// TIA Portal V20 export
FUNCTION_BLOCK "Sequence_3_JellyRollWinder"   // FB224, LAD
AUTHOR : ERsystem_FA2_DH. Kim
// stored: IsIECCheckEnabled true, MemoryReserve 100, Namespace Unit1.Em7, SetENOAutomatically false
   VAR
      statSelectedJobNumber { ExternalWritable := 'False'} : DInt;   // Evaluated Job Number
      instSequenceLADStatus { ExternalWritable := 'False'} : "LAF_StatusLadSequence";
      instSequenceLADControl { ExternalWritable := 'False'} : "LAF_ControlLadSequence";
      statTonTime { ExternalAccessible := 'False'; ExternalVisible := 'False'; ExternalWritable := 'False'} : Array[0..999] of TON_TIME;
   END_VAR
   VAR_TEMP
      tempCustomerAction : Bool;   // Placeholder for possible actions
      tempDo_nothing_and_wait_for_init : Bool;   // Placeholder for doing nothing
      tempSafeStateCondition : Bool;   // Temp Condition for the equipment module to be in a safe state
      tempIndex : Int;
   END_VAR
   VAR CONSTANT
      STEP_IDLE : DInt := 1;
      STEP_IMMEDIATE_STOP : DInt := 9001;   // Step executed when an immediate stop command is triggered for the sequence (i.e. when unit is in state aborting)
      JOB_1_STEP_01 : DInt := 101;
      JOB_1_STEP_10 : DInt := 110;
      JOB_1_STEP_20 : DInt := 120;
      JOB_1_STEP_30 : DInt := 130;
      JOB_1_STEP_80 : DInt := 180;
      JOB_1_STEP_90 : DInt := 190;
      JOB_2_STEP_01 : DInt := 201;
      JOB_2_STEP_10 : DInt := 210;
      JOB_2_STEP_20 : DInt := 220;
      JOB_2_STEP_21 : DInt := 221;
      JOB_2_STEP_90 : DInt := 290;
      JOB_3_STEP_01 : DInt := 301;
      JOB_3_STEP_10 : DInt := 310;
      JOB_3_STEP_11 : DInt := 311;
      JOB_3_STEP_12 : DInt := 312;
      JOB_3_STEP_13 : DInt := 313;
      JOB_3_STEP_90 : DInt := 390;
      JOB_4_STEP_01 : DInt := 401;
      JOB_4_STEP_10 : DInt := 410;
      JOB_4_STEP_20 : DInt := 420;
      JOB_4_STEP_21 : DInt := 421;
      JOB_4_STEP_90 : DInt := 490;
      JOB_5_STEP_01 : DInt := 501;
      JOB_5_STEP_10 : DInt := 510;
      JOB_5_STEP_11 : DInt := 511;
      JOB_5_STEP_20 : DInt := 520;
      JOB_5_STEP_21 : DInt := 521;
      JOB_5_STEP_90 : DInt := 590;
      JOB_6_STEP_01 : DInt := 601;
      JOB_6_STEP_10 : DInt := 610;
      JOB_6_STEP_20 : DInt := 620;
      JOB_6_STEP_21 : DInt := 621;
      JOB_6_STEP_30 : DInt := 630;
      JOB_6_STEP_80 : DInt := 680;
      JOB_6_STEP_81 : DInt := 681;
      JOB_6_STEP_90 : DInt := 690;
      JOB_7_STEP_01 : DInt := 701;
      JOB_7_STEP_10 : DInt := 710;
      JOB_7_STEP_20 : DInt := 720;
      JOB_7_STEP_30 : DInt := 730;
      JOB_7_STEP_40 : DInt := 740;
      JOB_7_STEP_50 : DInt := 750;
      JOB_7_STEP_90 : DInt := 790;
      JOB_10_STEP_01 : DInt := 1001;
      JOB_10_STEP_10 : DInt := 1010;
      JOB_10_STEP_90 : DInt := 1090;
      JOB_11_STEP_01 : DInt := 1101;
      JOB_11_STEP_10 : DInt := 1110;
      JOB_11_STEP_20 : DInt := 1120;
      JOB_11_STEP_90 : DInt := 1190;
      JOB_12_STEP_01 : DInt := 1201;
      JOB_12_STEP_10 : DInt := 1210;
      JOB_12_STEP_11 : DInt := 1211;
      JOB_12_STEP_90 : DInt := 1290;
      JOB_13_STEP_01 : DInt := 1301;
      JOB_13_STEP_10 : DInt := 1310;
      JOB_13_STEP_90 : DInt := 1390;
      JOB_14_STEP_01 : DInt := 1401;
      JOB_14_STEP_10 : DInt := 1410;
      JOB_14_STEP_90 : DInt := 1490;
      FALSE : Bool := FALSE;
      TRUE : Bool := TRUE;
   END_VAR
   VAR_TEMP   // added for the SCL form of the ladder/FBD networks
      _w1 : Bool;
      _w2 : Bool;
   END_VAR
BEGIN

REGION Network 1: BLOCK INFO HEADER
   // (company) / (C) Copyright (year)
   // ---------------------------------------------------------------------------------
   // Title:                             (Title of this block)
   // Comment/Function: (that is implemented in the block)
   // Library/Family:           (that the source is dedicated to)
   // Author:                        (department / person in charge / contact)
   // Target System:          (test system with FW version)
   // Engineering:              TIA Portal (SW version)
   // Restrictions:               (OB types, etc.)
   // Requirements:           (hardware, technological package, etc.)
   // ---------------------------------------------------------------------------------
   // Change log table:
   // Version          | Date             | Signature      | Expert in charge  | Changes applied ------------------------|----------------------|-------------------------|--------------------------------|-----------------------
   // 001.000.000 | yyyy-mm-dd | 0x00000000 | (name of expert) | First released version
END_REGION

REGION Network 2: DESCRIPTION
   // This is a template block provided by the Automation Framework. It can be used to create an own project.
   // The Block Info Header is prepared to put in your own data.
   // Description of the block could be added here and the docu created by Code2Docu.
END_REGION

REGION Network 3: ********************* CONTROL *************************
END_REGION

REGION Network 4: Sequence Control
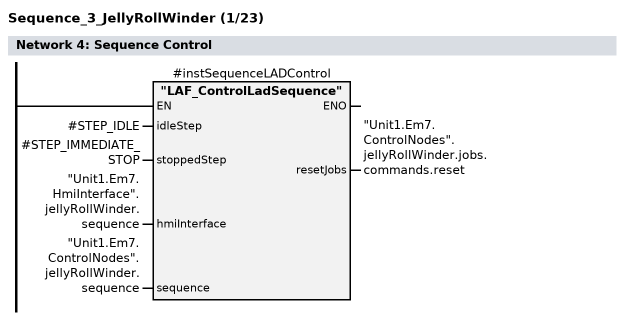
   RUNG wire#powerrail
      #instSequenceLADControl(idleStep := #STEP_IDLE, stoppedStep := #STEP_IMMEDIATE_STOP, hmiInterface := "Unit1.Em7.HmiInterface".jellyRollWinder.sequence, sequence := "Unit1.Em7.ControlNodes".jellyRollWinder.sequence, resetJobs => "Unit1.Em7.ControlNodes".jellyRollWinder.jobs.commands.reset)
   END_RUNG
   // the same network as SCL:
   #instSequenceLADControl(idleStep := #STEP_IDLE,   // "LAF_ControlLadSequence"
                           stoppedStep := #STEP_IMMEDIATE_STOP,
                           hmiInterface := "Unit1.Em7.HmiInterface".jellyRollWinder.sequence,
                           sequence := "Unit1.Em7.ControlNodes".jellyRollWinder.sequence,
                           resetJobs => "Unit1.Em7.ControlNodes".jellyRollWinder.jobs.commands.reset);
END_REGION

REGION Network 5: *************** JOB SELECT **************************
END_REGION

REGION Network 6: STEP IDLE
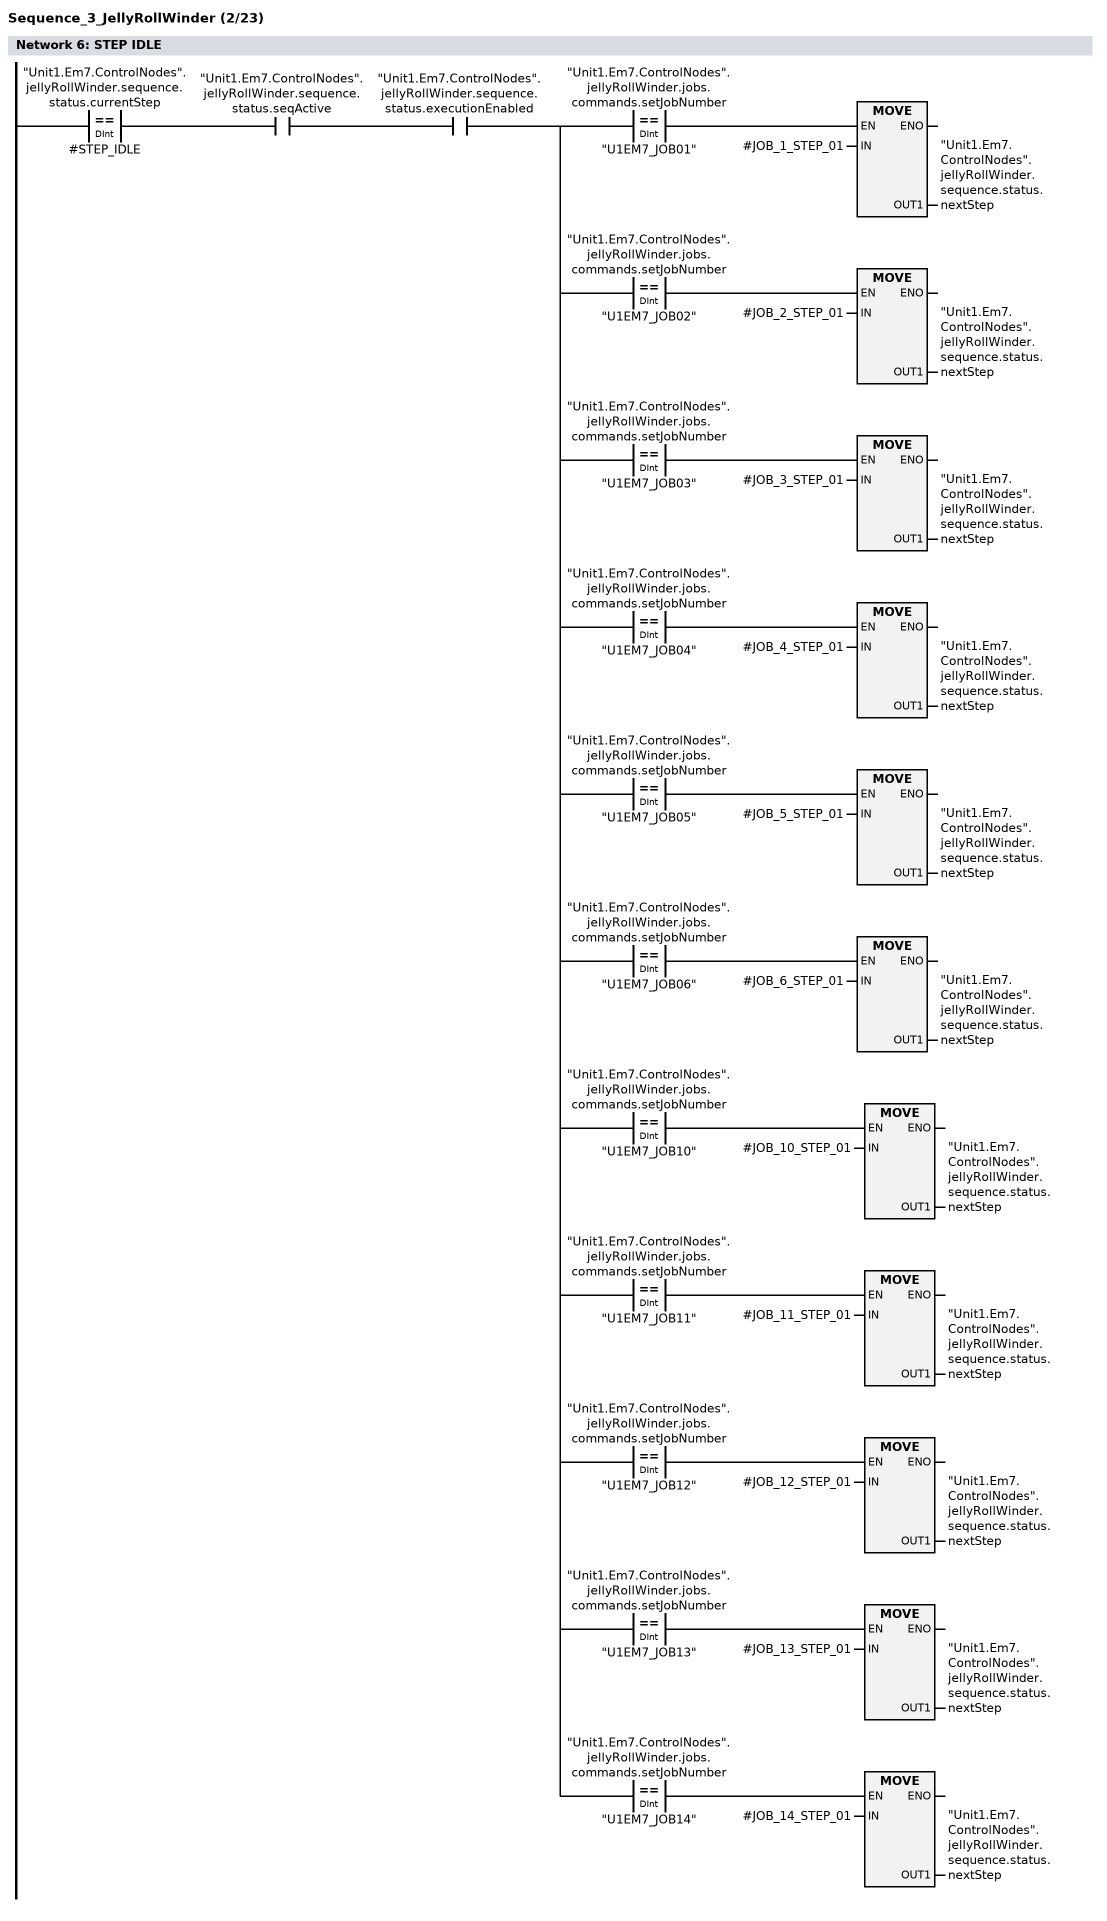
   RUNG wire#powerrail
      { S7_Templates := "SrcType := DInt" } EQ_Contact(in1 := "Unit1.Em7.ControlNodes".jellyRollWinder.sequence.status.currentStep, in2 := #STEP_IDLE)
      Contact( "Unit1.Em7.ControlNodes".jellyRollWinder.sequence.status.seqActive )
      Contact( "Unit1.Em7.ControlNodes".jellyRollWinder.sequence.status.executionEnabled )
      wire#w1
      { S7_Templates := "SrcType := DInt" } EQ_Contact(in1 := "Unit1.Em7.ControlNodes".jellyRollWinder.jobs.commands.setJobNumber, in2 := "U1EM7_JOB01")
      Move(in := #JOB_1_STEP_01, out1 => "Unit1.Em7.ControlNodes".jellyRollWinder.sequence.status.nextStep)
   END_RUNG
   RUNG wire#w1
      { S7_Templates := "SrcType := DInt" } EQ_Contact(in1 := "Unit1.Em7.ControlNodes".jellyRollWinder.jobs.commands.setJobNumber, in2 := "U1EM7_JOB02")
      Move(in := #JOB_2_STEP_01, out1 => "Unit1.Em7.ControlNodes".jellyRollWinder.sequence.status.nextStep)
   END_RUNG
   RUNG wire#w1
      { S7_Templates := "SrcType := DInt" } EQ_Contact(in1 := "Unit1.Em7.ControlNodes".jellyRollWinder.jobs.commands.setJobNumber, in2 := "U1EM7_JOB03")
      Move(in := #JOB_3_STEP_01, out1 => "Unit1.Em7.ControlNodes".jellyRollWinder.sequence.status.nextStep)
   END_RUNG
   RUNG wire#w1
      { S7_Templates := "SrcType := DInt" } EQ_Contact(in1 := "Unit1.Em7.ControlNodes".jellyRollWinder.jobs.commands.setJobNumber, in2 := "U1EM7_JOB04")
      Move(in := #JOB_4_STEP_01, out1 => "Unit1.Em7.ControlNodes".jellyRollWinder.sequence.status.nextStep)
   END_RUNG
   RUNG wire#w1
      { S7_Templates := "SrcType := DInt" } EQ_Contact(in1 := "Unit1.Em7.ControlNodes".jellyRollWinder.jobs.commands.setJobNumber, in2 := "U1EM7_JOB05")
      Move(in := #JOB_5_STEP_01, out1 => "Unit1.Em7.ControlNodes".jellyRollWinder.sequence.status.nextStep)
   END_RUNG
   RUNG wire#w1
      { S7_Templates := "SrcType := DInt" } EQ_Contact(in1 := "Unit1.Em7.ControlNodes".jellyRollWinder.jobs.commands.setJobNumber, in2 := "U1EM7_JOB06")
      Move(in := #JOB_6_STEP_01, out1 => "Unit1.Em7.ControlNodes".jellyRollWinder.sequence.status.nextStep)
   END_RUNG
   RUNG wire#w1
      { S7_Templates := "SrcType := DInt" } EQ_Contact(in1 := "Unit1.Em7.ControlNodes".jellyRollWinder.jobs.commands.setJobNumber, in2 := "U1EM7_JOB10")
      Move(in := #JOB_10_STEP_01, out1 => "Unit1.Em7.ControlNodes".jellyRollWinder.sequence.status.nextStep)
   END_RUNG
   RUNG wire#w1
      { S7_Templates := "SrcType := DInt" } EQ_Contact(in1 := "Unit1.Em7.ControlNodes".jellyRollWinder.jobs.commands.setJobNumber, in2 := "U1EM7_JOB11")
      Move(in := #JOB_11_STEP_01, out1 => "Unit1.Em7.ControlNodes".jellyRollWinder.sequence.status.nextStep)
   END_RUNG
   RUNG wire#w1
      { S7_Templates := "SrcType := DInt" } EQ_Contact(in1 := "Unit1.Em7.ControlNodes".jellyRollWinder.jobs.commands.setJobNumber, in2 := "U1EM7_JOB12")
      Move(in := #JOB_12_STEP_01, out1 => "Unit1.Em7.ControlNodes".jellyRollWinder.sequence.status.nextStep)
   END_RUNG
   RUNG wire#w1
      { S7_Templates := "SrcType := DInt" } EQ_Contact(in1 := "Unit1.Em7.ControlNodes".jellyRollWinder.jobs.commands.setJobNumber, in2 := "U1EM7_JOB13")
      Move(in := #JOB_13_STEP_01, out1 => "Unit1.Em7.ControlNodes".jellyRollWinder.sequence.status.nextStep)
   END_RUNG
   RUNG wire#w1
      { S7_Templates := "SrcType := DInt" } EQ_Contact(in1 := "Unit1.Em7.ControlNodes".jellyRollWinder.jobs.commands.setJobNumber, in2 := "U1EM7_JOB14")
      Move(in := #JOB_14_STEP_01, out1 => "Unit1.Em7.ControlNodes".jellyRollWinder.sequence.status.nextStep)
   END_RUNG
   // the same network as SCL:
   #_w1 := ("Unit1.Em7.ControlNodes".jellyRollWinder.sequence.status.currentStep = #STEP_IDLE) AND "Unit1.Em7.ControlNodes".jellyRollWinder.sequence.status.seqActive AND "Unit1.Em7.ControlNodes".jellyRollWinder.sequence.status.executionEnabled;
   IF #_w1 AND ("Unit1.Em7.ControlNodes".jellyRollWinder.jobs.commands.setJobNumber = "U1EM7_JOB01") THEN
       "Unit1.Em7.ControlNodes".jellyRollWinder.sequence.status.nextStep := #JOB_1_STEP_01;
   END_IF;
   IF #_w1 AND ("Unit1.Em7.ControlNodes".jellyRollWinder.jobs.commands.setJobNumber = "U1EM7_JOB02") THEN
       "Unit1.Em7.ControlNodes".jellyRollWinder.sequence.status.nextStep := #JOB_2_STEP_01;
   END_IF;
   IF #_w1 AND ("Unit1.Em7.ControlNodes".jellyRollWinder.jobs.commands.setJobNumber = "U1EM7_JOB03") THEN
       "Unit1.Em7.ControlNodes".jellyRollWinder.sequence.status.nextStep := #JOB_3_STEP_01;
   END_IF;
   IF #_w1 AND ("Unit1.Em7.ControlNodes".jellyRollWinder.jobs.commands.setJobNumber = "U1EM7_JOB04") THEN
       "Unit1.Em7.ControlNodes".jellyRollWinder.sequence.status.nextStep := #JOB_4_STEP_01;
   END_IF;
   IF #_w1 AND ("Unit1.Em7.ControlNodes".jellyRollWinder.jobs.commands.setJobNumber = "U1EM7_JOB05") THEN
       "Unit1.Em7.ControlNodes".jellyRollWinder.sequence.status.nextStep := #JOB_5_STEP_01;
   END_IF;
   IF #_w1 AND ("Unit1.Em7.ControlNodes".jellyRollWinder.jobs.commands.setJobNumber = "U1EM7_JOB06") THEN
       "Unit1.Em7.ControlNodes".jellyRollWinder.sequence.status.nextStep := #JOB_6_STEP_01;
   END_IF;
   IF #_w1 AND ("Unit1.Em7.ControlNodes".jellyRollWinder.jobs.commands.setJobNumber = "U1EM7_JOB10") THEN
       "Unit1.Em7.ControlNodes".jellyRollWinder.sequence.status.nextStep := #JOB_10_STEP_01;
   END_IF;
   IF #_w1 AND ("Unit1.Em7.ControlNodes".jellyRollWinder.jobs.commands.setJobNumber = "U1EM7_JOB11") THEN
       "Unit1.Em7.ControlNodes".jellyRollWinder.sequence.status.nextStep := #JOB_11_STEP_01;
   END_IF;
   IF #_w1 AND ("Unit1.Em7.ControlNodes".jellyRollWinder.jobs.commands.setJobNumber = "U1EM7_JOB12") THEN
       "Unit1.Em7.ControlNodes".jellyRollWinder.sequence.status.nextStep := #JOB_12_STEP_01;
   END_IF;
   IF #_w1 AND ("Unit1.Em7.ControlNodes".jellyRollWinder.jobs.commands.setJobNumber = "U1EM7_JOB13") THEN
       "Unit1.Em7.ControlNodes".jellyRollWinder.sequence.status.nextStep := #JOB_13_STEP_01;
   END_IF;
   IF #_w1 AND ("Unit1.Em7.ControlNodes".jellyRollWinder.jobs.commands.setJobNumber = "U1EM7_JOB14") THEN
       "Unit1.Em7.ControlNodes".jellyRollWinder.sequence.status.nextStep := #JOB_14_STEP_01;
   END_IF;
END_REGION

REGION Network 7: ******************** JOB[1] EM HOMING ********************
END_REGION

REGION Network 8: Step[101] : JOB[1] Condition
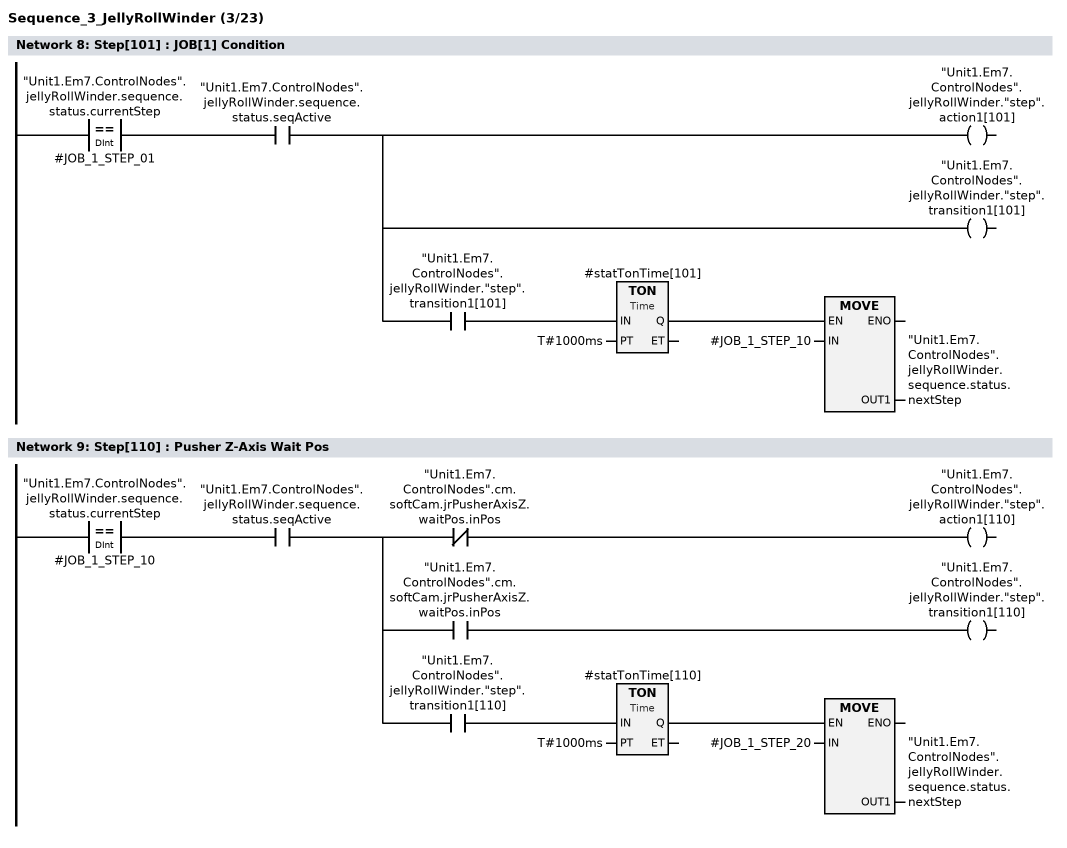
   RUNG wire#powerrail
      { S7_Templates := "SrcType := DInt" } EQ_Contact(in1 := "Unit1.Em7.ControlNodes".jellyRollWinder.sequence.status.currentStep, in2 := #JOB_1_STEP_01)
      Contact( "Unit1.Em7.ControlNodes".jellyRollWinder.sequence.status.seqActive )
      wire#w1
      Coil( "Unit1.Em7.ControlNodes".jellyRollWinder."step".action1[101] )
   END_RUNG
   RUNG wire#w1
      Coil( "Unit1.Em7.ControlNodes".jellyRollWinder."step".transition1[101] )
   END_RUNG
   RUNG wire#w1
      Contact( "Unit1.Em7.ControlNodes".jellyRollWinder."step".transition1[101] )
      { S7_Templates := "time_type := Time" } #statTonTime[101].TON(pt := T#1000ms, et =>)
      Move(in := #JOB_1_STEP_10, out1 => "Unit1.Em7.ControlNodes".jellyRollWinder.sequence.status.nextStep)
   END_RUNG
   // the same network as SCL:
   "Unit1.Em7.ControlNodes".jellyRollWinder."step".action1[101] := ("Unit1.Em7.ControlNodes".jellyRollWinder.sequence.status.currentStep = #JOB_1_STEP_01) AND "Unit1.Em7.ControlNodes".jellyRollWinder.sequence.status.seqActive;
   "Unit1.Em7.ControlNodes".jellyRollWinder."step".transition1[101] := ("Unit1.Em7.ControlNodes".jellyRollWinder.sequence.status.currentStep = #JOB_1_STEP_01) AND "Unit1.Em7.ControlNodes".jellyRollWinder.sequence.status.seqActive;
   #statTonTime[101].TON(IN := ("Unit1.Em7.ControlNodes".jellyRollWinder.sequence.status.currentStep = #JOB_1_STEP_01) AND "Unit1.Em7.ControlNodes".jellyRollWinder.sequence.status.seqActive AND "Unit1.Em7.ControlNodes".jellyRollWinder."step".transition1[101],
                         PT := T#1000ms);
   IF #statTonTime[101].Q THEN
       "Unit1.Em7.ControlNodes".jellyRollWinder.sequence.status.nextStep := #JOB_1_STEP_10;
   END_IF;
END_REGION

REGION Network 9: Step[110] : Pusher Z-Axis Wait Pos
   RUNG wire#powerrail
      { S7_Templates := "SrcType := DInt" } EQ_Contact(in1 := "Unit1.Em7.ControlNodes".jellyRollWinder.sequence.status.currentStep, in2 := #JOB_1_STEP_10)
      Contact( "Unit1.Em7.ControlNodes".jellyRollWinder.sequence.status.seqActive )
      wire#w1
      I_Contact( "Unit1.Em7.ControlNodes".cm.softCam.jrPusherAxisZ.waitPos.inPos )
      Coil( "Unit1.Em7.ControlNodes".jellyRollWinder."step".action1[110] )
   END_RUNG
   RUNG wire#w1
      Contact( "Unit1.Em7.ControlNodes".cm.softCam.jrPusherAxisZ.waitPos.inPos )
      Coil( "Unit1.Em7.ControlNodes".jellyRollWinder."step".transition1[110] )
   END_RUNG
   RUNG wire#w1
      Contact( "Unit1.Em7.ControlNodes".jellyRollWinder."step".transition1[110] )
      { S7_Templates := "time_type := Time" } #statTonTime[110].TON(pt := T#1000ms, et =>)
      Move(in := #JOB_1_STEP_20, out1 => "Unit1.Em7.ControlNodes".jellyRollWinder.sequence.status.nextStep)
   END_RUNG
   // the same network as SCL:
   #_w1 := ("Unit1.Em7.ControlNodes".jellyRollWinder.sequence.status.currentStep = #JOB_1_STEP_10) AND "Unit1.Em7.ControlNodes".jellyRollWinder.sequence.status.seqActive;
   "Unit1.Em7.ControlNodes".jellyRollWinder."step".action1[110] := #_w1 AND NOT "Unit1.Em7.ControlNodes".cm.softCam.jrPusherAxisZ.waitPos.inPos;
   "Unit1.Em7.ControlNodes".jellyRollWinder."step".transition1[110] := #_w1 AND "Unit1.Em7.ControlNodes".cm.softCam.jrPusherAxisZ.waitPos.inPos;
   #statTonTime[110].TON(IN := #_w1 AND "Unit1.Em7.ControlNodes".jellyRollWinder."step".transition1[110],
                         PT := T#1000ms);
   IF #statTonTime[110].Q THEN
       "Unit1.Em7.ControlNodes".jellyRollWinder.sequence.status.nextStep := #JOB_1_STEP_20;
   END_IF;
END_REGION

REGION Network 10: Step[120]: Pusher Backward
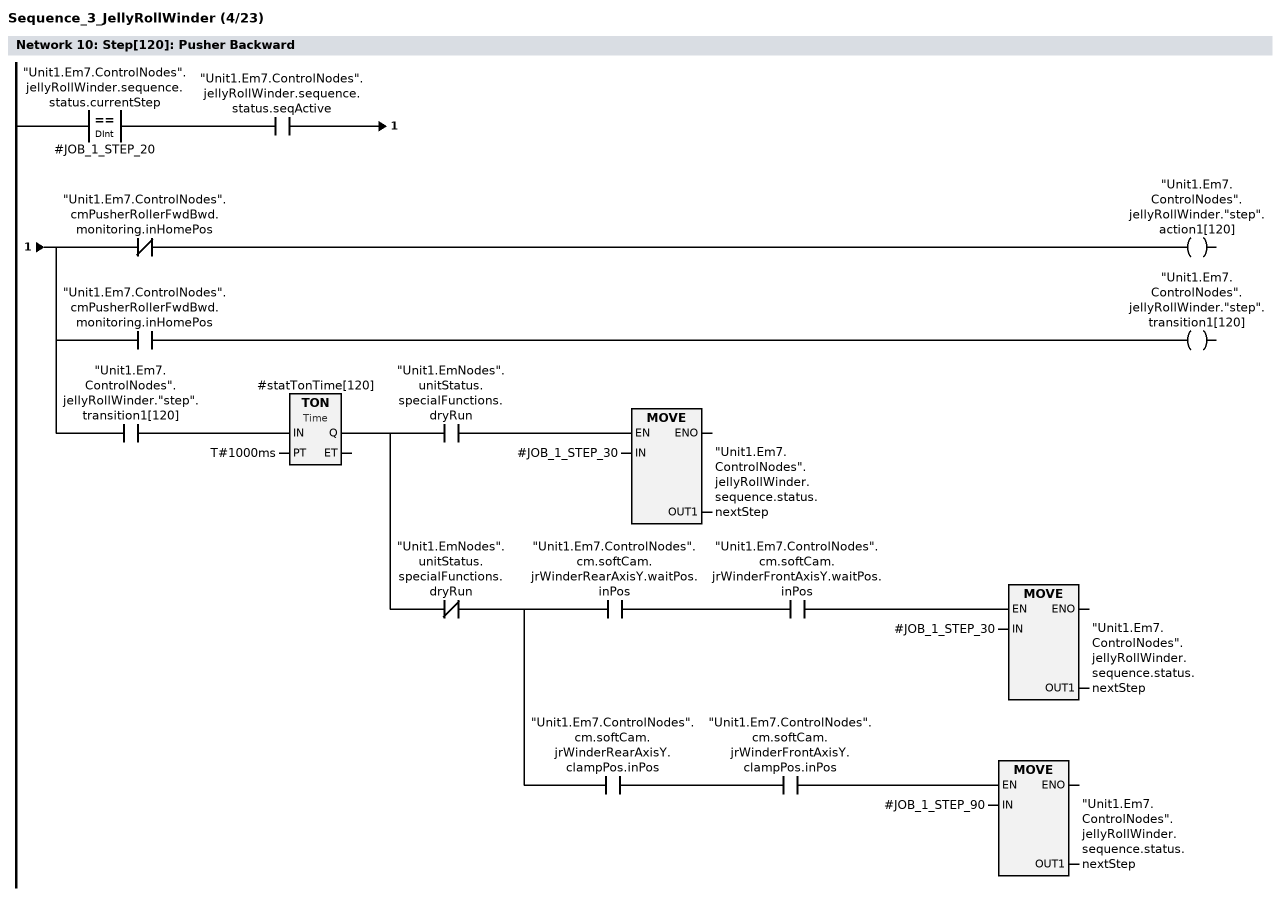
   RUNG wire#powerrail
      { S7_Templates := "SrcType := DInt" } EQ_Contact(in1 := "Unit1.Em7.ControlNodes".jellyRollWinder.sequence.status.currentStep, in2 := #JOB_1_STEP_20)
      Contact( "Unit1.Em7.ControlNodes".jellyRollWinder.sequence.status.seqActive )
      wire#w1
      I_Contact( "Unit1.Em7.ControlNodes".cmPusherRollerFwdBwd.monitoring.inHomePos )
      Coil( "Unit1.Em7.ControlNodes".jellyRollWinder."step".action1[120] )
   END_RUNG
   RUNG wire#w1
      Contact( "Unit1.Em7.ControlNodes".cmPusherRollerFwdBwd.monitoring.inHomePos )
      Coil( "Unit1.Em7.ControlNodes".jellyRollWinder."step".transition1[120] )
   END_RUNG
   RUNG wire#w1
      Contact( "Unit1.Em7.ControlNodes".jellyRollWinder."step".transition1[120] )
      { S7_Templates := "time_type := Time" } #statTonTime[120].TON(pt := T#1000ms, et =>)
      wire#w2
      Contact( "Unit1.EmNodes".unitStatus.specialFunctions.dryRun )
      Move(in := #JOB_1_STEP_30, out1 => "Unit1.Em7.ControlNodes".jellyRollWinder.sequence.status.nextStep)
   END_RUNG
   RUNG wire#w2
      I_Contact( "Unit1.EmNodes".unitStatus.specialFunctions.dryRun )
      wire#w3
      Contact( "Unit1.Em7.ControlNodes".cm.softCam.jrWinderRearAxisY.waitPos.inPos )
      Contact( "Unit1.Em7.ControlNodes".cm.softCam.jrWinderFrontAxisY.waitPos.inPos )
      Move(in := #JOB_1_STEP_30, out1 => "Unit1.Em7.ControlNodes".jellyRollWinder.sequence.status.nextStep)
   END_RUNG
   RUNG wire#w3
      Contact( "Unit1.Em7.ControlNodes".cm.softCam.jrWinderRearAxisY.clampPos.inPos )
      Contact( "Unit1.Em7.ControlNodes".cm.softCam.jrWinderFrontAxisY.clampPos.inPos )
      Move(in := #JOB_1_STEP_90, out1 => "Unit1.Em7.ControlNodes".jellyRollWinder.sequence.status.nextStep)
   END_RUNG
   // the same network as SCL:
   #_w1 := ("Unit1.Em7.ControlNodes".jellyRollWinder.sequence.status.currentStep = #JOB_1_STEP_20) AND "Unit1.Em7.ControlNodes".jellyRollWinder.sequence.status.seqActive;
   "Unit1.Em7.ControlNodes".jellyRollWinder."step".action1[120] := #_w1 AND NOT "Unit1.Em7.ControlNodes".cmPusherRollerFwdBwd.monitoring.inHomePos;
   "Unit1.Em7.ControlNodes".jellyRollWinder."step".transition1[120] := #_w1 AND "Unit1.Em7.ControlNodes".cmPusherRollerFwdBwd.monitoring.inHomePos;
   #statTonTime[120].TON(IN := #_w1 AND "Unit1.Em7.ControlNodes".jellyRollWinder."step".transition1[120],
                         PT := T#1000ms);
   IF #statTonTime[120].Q AND "Unit1.EmNodes".unitStatus.specialFunctions.dryRun THEN
       "Unit1.Em7.ControlNodes".jellyRollWinder.sequence.status.nextStep := #JOB_1_STEP_30;
   END_IF;
   #_w2 := #statTonTime[120].Q AND NOT "Unit1.EmNodes".unitStatus.specialFunctions.dryRun;
   IF #_w2 AND "Unit1.Em7.ControlNodes".cm.softCam.jrWinderRearAxisY.waitPos.inPos AND "Unit1.Em7.ControlNodes".cm.softCam.jrWinderFrontAxisY.waitPos.inPos THEN
       "Unit1.Em7.ControlNodes".jellyRollWinder.sequence.status.nextStep := #JOB_1_STEP_30;
   END_IF;
   IF #_w2 AND "Unit1.Em7.ControlNodes".cm.softCam.jrWinderRearAxisY.clampPos.inPos AND "Unit1.Em7.ControlNodes".cm.softCam.jrWinderFrontAxisY.clampPos.inPos THEN
       "Unit1.Em7.ControlNodes".jellyRollWinder.sequence.status.nextStep := #JOB_1_STEP_90;
   END_IF;
END_REGION

REGION Network 11: Step[130] : Winder Open
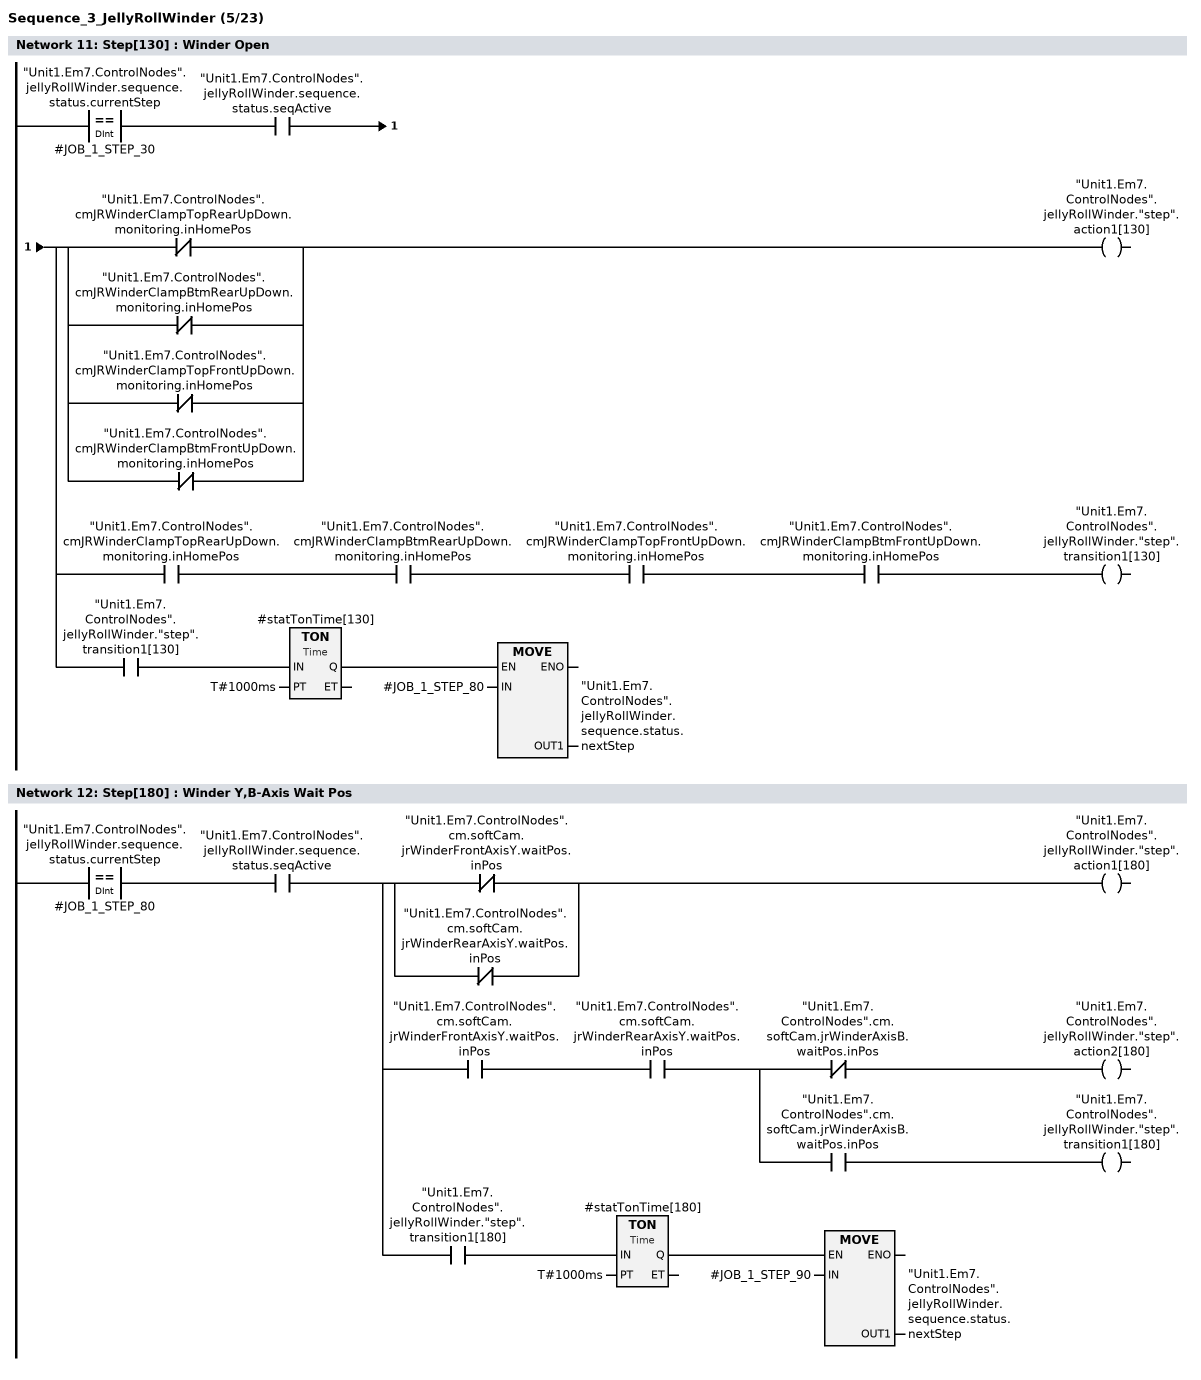
   RUNG wire#powerrail
      { S7_Templates := "SrcType := DInt" } EQ_Contact(in1 := "Unit1.Em7.ControlNodes".jellyRollWinder.sequence.status.currentStep, in2 := #JOB_1_STEP_30)
      Contact( "Unit1.Em7.ControlNodes".jellyRollWinder.sequence.status.seqActive )
      wire#w1
      I_Contact( "Unit1.Em7.ControlNodes".cmJRWinderClampTopRearUpDown.monitoring.inHomePos )
      wire#w2
      Coil( "Unit1.Em7.ControlNodes".jellyRollWinder."step".action1[130] )
   END_RUNG
   RUNG wire#w1
      I_Contact( "Unit1.Em7.ControlNodes".cmJRWinderClampBtmRearUpDown.monitoring.inHomePos )
   END_RUNG wire#w2
   RUNG wire#w1
      I_Contact( "Unit1.Em7.ControlNodes".cmJRWinderClampTopFrontUpDown.monitoring.inHomePos )
   END_RUNG wire#w2
   RUNG wire#w1
      I_Contact( "Unit1.Em7.ControlNodes".cmJRWinderClampBtmFrontUpDown.monitoring.inHomePos )
   END_RUNG wire#w2
   RUNG wire#w1
      Contact( "Unit1.Em7.ControlNodes".cmJRWinderClampTopRearUpDown.monitoring.inHomePos )
      Contact( "Unit1.Em7.ControlNodes".cmJRWinderClampBtmRearUpDown.monitoring.inHomePos )
      Contact( "Unit1.Em7.ControlNodes".cmJRWinderClampTopFrontUpDown.monitoring.inHomePos )
      Contact( "Unit1.Em7.ControlNodes".cmJRWinderClampBtmFrontUpDown.monitoring.inHomePos )
      Coil( "Unit1.Em7.ControlNodes".jellyRollWinder."step".transition1[130] )
   END_RUNG
   RUNG wire#w1
      Contact( "Unit1.Em7.ControlNodes".jellyRollWinder."step".transition1[130] )
      { S7_Templates := "time_type := Time" } #statTonTime[130].TON(pt := T#1000ms, et =>)
      Move(in := #JOB_1_STEP_80, out1 => "Unit1.Em7.ControlNodes".jellyRollWinder.sequence.status.nextStep)
   END_RUNG
   // the same network as SCL:
   #_w1 := ("Unit1.Em7.ControlNodes".jellyRollWinder.sequence.status.currentStep = #JOB_1_STEP_30) AND "Unit1.Em7.ControlNodes".jellyRollWinder.sequence.status.seqActive;
   "Unit1.Em7.ControlNodes".jellyRollWinder."step".action1[130] := #_w1 AND (NOT "Unit1.Em7.ControlNodes".cmJRWinderClampTopRearUpDown.monitoring.inHomePos OR NOT "Unit1.Em7.ControlNodes".cmJRWinderClampBtmRearUpDown.monitoring.inHomePos OR NOT "Unit1.Em7.ControlNodes".cmJRWinderClampTopFrontUpDown.monitoring.inHomePos OR NOT "Unit1.Em7.ControlNodes".cmJRWinderClampBtmFrontUpDown.monitoring.inHomePos);
   "Unit1.Em7.ControlNodes".jellyRollWinder."step".transition1[130] := #_w1 AND "Unit1.Em7.ControlNodes".cmJRWinderClampTopRearUpDown.monitoring.inHomePos AND "Unit1.Em7.ControlNodes".cmJRWinderClampBtmRearUpDown.monitoring.inHomePos AND "Unit1.Em7.ControlNodes".cmJRWinderClampTopFrontUpDown.monitoring.inHomePos AND "Unit1.Em7.ControlNodes".cmJRWinderClampBtmFrontUpDown.monitoring.inHomePos;
   #statTonTime[130].TON(IN := #_w1 AND "Unit1.Em7.ControlNodes".jellyRollWinder."step".transition1[130],
                         PT := T#1000ms);
   IF #statTonTime[130].Q THEN
       "Unit1.Em7.ControlNodes".jellyRollWinder.sequence.status.nextStep := #JOB_1_STEP_80;
   END_IF;
END_REGION

REGION Network 12: Step[180] : Winder Y,B-Axis Wait Pos
   RUNG wire#powerrail
      { S7_Templates := "SrcType := DInt" } EQ_Contact(in1 := "Unit1.Em7.ControlNodes".jellyRollWinder.sequence.status.currentStep, in2 := #JOB_1_STEP_80)
      Contact( "Unit1.Em7.ControlNodes".jellyRollWinder.sequence.status.seqActive )
      wire#w1
      I_Contact( "Unit1.Em7.ControlNodes".cm.softCam.jrWinderFrontAxisY.waitPos.inPos )
      wire#w2
      Coil( "Unit1.Em7.ControlNodes".jellyRollWinder."step".action1[180] )
   END_RUNG
   RUNG wire#w1
      I_Contact( "Unit1.Em7.ControlNodes".cm.softCam.jrWinderRearAxisY.waitPos.inPos )
   END_RUNG wire#w2
   RUNG wire#w1
      Contact( "Unit1.Em7.ControlNodes".cm.softCam.jrWinderFrontAxisY.waitPos.inPos )
      Contact( "Unit1.Em7.ControlNodes".cm.softCam.jrWinderRearAxisY.waitPos.inPos )
      wire#w3
      I_Contact( "Unit1.Em7.ControlNodes".cm.softCam.jrWinderAxisB.waitPos.inPos )
      Coil( "Unit1.Em7.ControlNodes".jellyRollWinder."step".action2[180] )
   END_RUNG
   RUNG wire#w3
      Contact( "Unit1.Em7.ControlNodes".cm.softCam.jrWinderAxisB.waitPos.inPos )
      Coil( "Unit1.Em7.ControlNodes".jellyRollWinder."step".transition1[180] )
   END_RUNG
   RUNG wire#w1
      Contact( "Unit1.Em7.ControlNodes".jellyRollWinder."step".transition1[180] )
      { S7_Templates := "time_type := Time" } #statTonTime[180].TON(pt := T#1000ms, et =>)
      Move(in := #JOB_1_STEP_90, out1 => "Unit1.Em7.ControlNodes".jellyRollWinder.sequence.status.nextStep)
   END_RUNG
   // the same network as SCL:
   #_w1 := ("Unit1.Em7.ControlNodes".jellyRollWinder.sequence.status.currentStep = #JOB_1_STEP_80) AND "Unit1.Em7.ControlNodes".jellyRollWinder.sequence.status.seqActive;
   "Unit1.Em7.ControlNodes".jellyRollWinder."step".action1[180] := #_w1 AND (NOT "Unit1.Em7.ControlNodes".cm.softCam.jrWinderFrontAxisY.waitPos.inPos OR NOT "Unit1.Em7.ControlNodes".cm.softCam.jrWinderRearAxisY.waitPos.inPos);
   #_w2 := #_w1 AND "Unit1.Em7.ControlNodes".cm.softCam.jrWinderFrontAxisY.waitPos.inPos AND "Unit1.Em7.ControlNodes".cm.softCam.jrWinderRearAxisY.waitPos.inPos;
   "Unit1.Em7.ControlNodes".jellyRollWinder."step".action2[180] := #_w2 AND NOT "Unit1.Em7.ControlNodes".cm.softCam.jrWinderAxisB.waitPos.inPos;
   "Unit1.Em7.ControlNodes".jellyRollWinder."step".transition1[180] := #_w2 AND "Unit1.Em7.ControlNodes".cm.softCam.jrWinderAxisB.waitPos.inPos;
   #statTonTime[180].TON(IN := #_w1 AND "Unit1.Em7.ControlNodes".jellyRollWinder."step".transition1[180],
                         PT := T#1000ms);
   IF #statTonTime[180].Q THEN
       "Unit1.Em7.ControlNodes".jellyRollWinder.sequence.status.nextStep := #JOB_1_STEP_90;
   END_IF;
END_REGION

REGION Network 13: Step[190] : Job[1] Step End
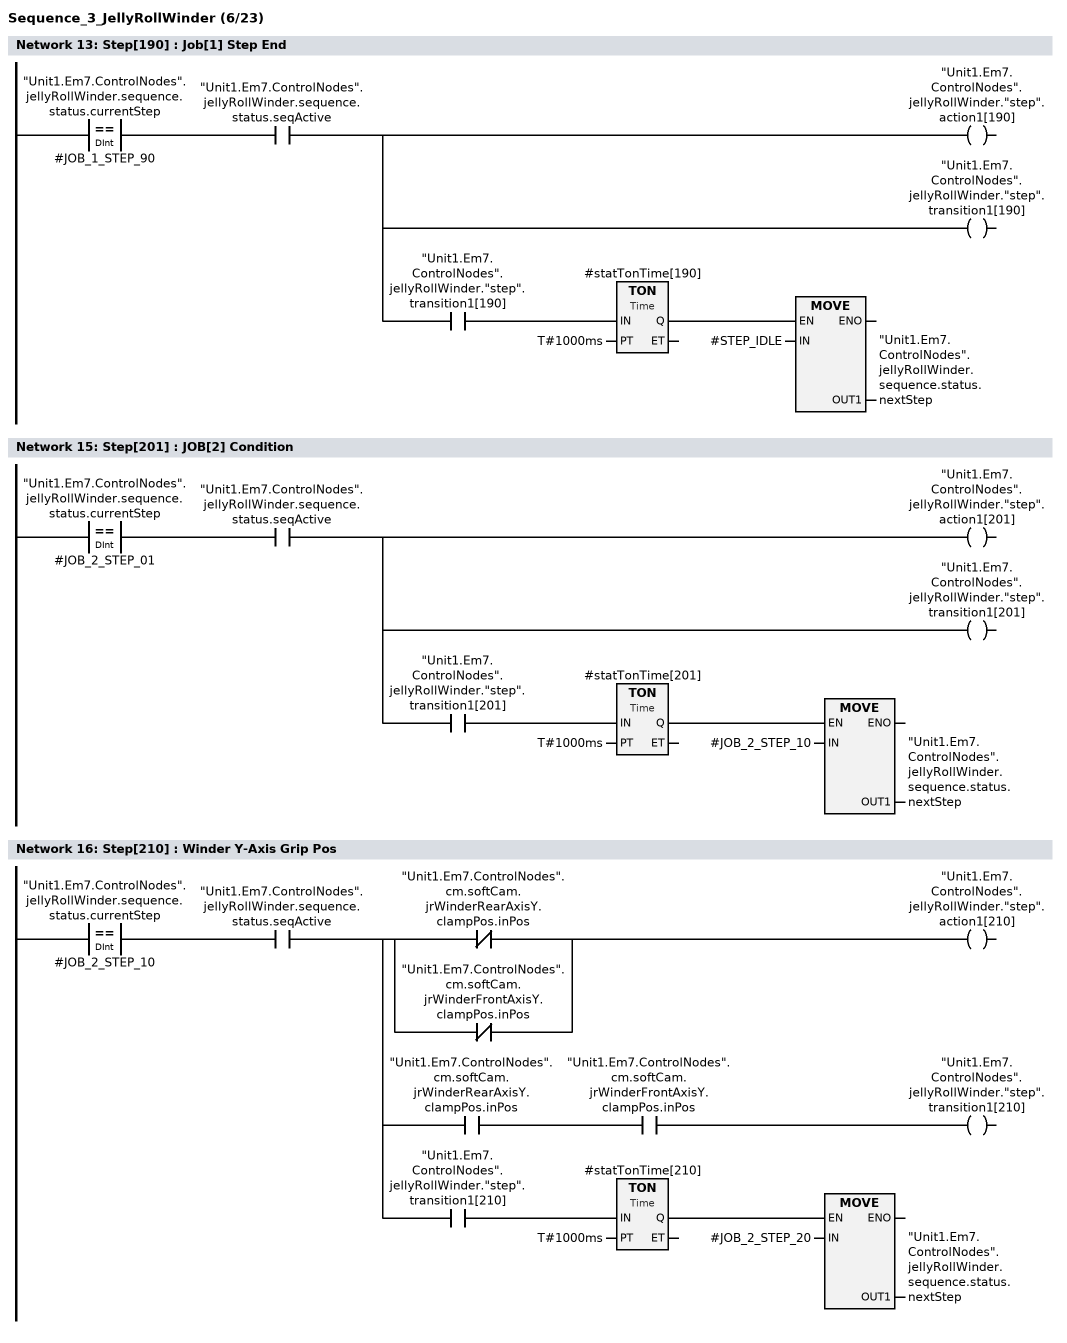
   RUNG wire#powerrail
      { S7_Templates := "SrcType := DInt" } EQ_Contact(in1 := "Unit1.Em7.ControlNodes".jellyRollWinder.sequence.status.currentStep, in2 := #JOB_1_STEP_90)
      Contact( "Unit1.Em7.ControlNodes".jellyRollWinder.sequence.status.seqActive )
      wire#w1
      Coil( "Unit1.Em7.ControlNodes".jellyRollWinder."step".action1[190] )
   END_RUNG
   RUNG wire#w1
      Coil( "Unit1.Em7.ControlNodes".jellyRollWinder."step".transition1[190] )
   END_RUNG
   RUNG wire#w1
      Contact( "Unit1.Em7.ControlNodes".jellyRollWinder."step".transition1[190] )
      { S7_Templates := "time_type := Time" } #statTonTime[190].TON(pt := T#1000ms, et =>)
      Move(in := #STEP_IDLE, out1 => "Unit1.Em7.ControlNodes".jellyRollWinder.sequence.status.nextStep)
   END_RUNG
   // the same network as SCL:
   "Unit1.Em7.ControlNodes".jellyRollWinder."step".action1[190] := ("Unit1.Em7.ControlNodes".jellyRollWinder.sequence.status.currentStep = #JOB_1_STEP_90) AND "Unit1.Em7.ControlNodes".jellyRollWinder.sequence.status.seqActive;
   "Unit1.Em7.ControlNodes".jellyRollWinder."step".transition1[190] := ("Unit1.Em7.ControlNodes".jellyRollWinder.sequence.status.currentStep = #JOB_1_STEP_90) AND "Unit1.Em7.ControlNodes".jellyRollWinder.sequence.status.seqActive;
   #statTonTime[190].TON(IN := ("Unit1.Em7.ControlNodes".jellyRollWinder.sequence.status.currentStep = #JOB_1_STEP_90) AND "Unit1.Em7.ControlNodes".jellyRollWinder.sequence.status.seqActive AND "Unit1.Em7.ControlNodes".jellyRollWinder."step".transition1[190],
                         PT := T#1000ms);
   IF #statTonTime[190].Q THEN
       "Unit1.Em7.ControlNodes".jellyRollWinder.sequence.status.nextStep := #STEP_IDLE;
   END_IF;
END_REGION

REGION Network 14: ******************** JOB[2] Load ********************
END_REGION

REGION Network 15: Step[201] : JOB[2] Condition
   RUNG wire#powerrail
      { S7_Templates := "SrcType := DInt" } EQ_Contact(in1 := "Unit1.Em7.ControlNodes".jellyRollWinder.sequence.status.currentStep, in2 := #JOB_2_STEP_01)
      Contact( "Unit1.Em7.ControlNodes".jellyRollWinder.sequence.status.seqActive )
      wire#w1
      Coil( "Unit1.Em7.ControlNodes".jellyRollWinder."step".action1[201] )
   END_RUNG
   RUNG wire#w1
      Coil( "Unit1.Em7.ControlNodes".jellyRollWinder."step".transition1[201] )
   END_RUNG
   RUNG wire#w1
      Contact( "Unit1.Em7.ControlNodes".jellyRollWinder."step".transition1[201] )
      { S7_Templates := "time_type := Time" } #statTonTime[201].TON(pt := T#1000ms, et =>)
      Move(in := #JOB_2_STEP_10, out1 => "Unit1.Em7.ControlNodes".jellyRollWinder.sequence.status.nextStep)
   END_RUNG
   // the same network as SCL:
   "Unit1.Em7.ControlNodes".jellyRollWinder."step".action1[201] := ("Unit1.Em7.ControlNodes".jellyRollWinder.sequence.status.currentStep = #JOB_2_STEP_01) AND "Unit1.Em7.ControlNodes".jellyRollWinder.sequence.status.seqActive;
   "Unit1.Em7.ControlNodes".jellyRollWinder."step".transition1[201] := ("Unit1.Em7.ControlNodes".jellyRollWinder.sequence.status.currentStep = #JOB_2_STEP_01) AND "Unit1.Em7.ControlNodes".jellyRollWinder.sequence.status.seqActive;
   #statTonTime[201].TON(IN := ("Unit1.Em7.ControlNodes".jellyRollWinder.sequence.status.currentStep = #JOB_2_STEP_01) AND "Unit1.Em7.ControlNodes".jellyRollWinder.sequence.status.seqActive AND "Unit1.Em7.ControlNodes".jellyRollWinder."step".transition1[201],
                         PT := T#1000ms);
   IF #statTonTime[201].Q THEN
       "Unit1.Em7.ControlNodes".jellyRollWinder.sequence.status.nextStep := #JOB_2_STEP_10;
   END_IF;
END_REGION

REGION Network 16: Step[210] : Winder Y-Axis Grip Pos
   RUNG wire#powerrail
      { S7_Templates := "SrcType := DInt" } EQ_Contact(in1 := "Unit1.Em7.ControlNodes".jellyRollWinder.sequence.status.currentStep, in2 := #JOB_2_STEP_10)
      Contact( "Unit1.Em7.ControlNodes".jellyRollWinder.sequence.status.seqActive )
      wire#w1
      I_Contact( "Unit1.Em7.ControlNodes".cm.softCam.jrWinderRearAxisY.clampPos.inPos )
      wire#w2
      Coil( "Unit1.Em7.ControlNodes".jellyRollWinder."step".action1[210] )
   END_RUNG
   RUNG wire#w1
      I_Contact( "Unit1.Em7.ControlNodes".cm.softCam.jrWinderFrontAxisY.clampPos.inPos )
   END_RUNG wire#w2
   RUNG wire#w1
      Contact( "Unit1.Em7.ControlNodes".cm.softCam.jrWinderRearAxisY.clampPos.inPos )
      Contact( "Unit1.Em7.ControlNodes".cm.softCam.jrWinderFrontAxisY.clampPos.inPos )
      Coil( "Unit1.Em7.ControlNodes".jellyRollWinder."step".transition1[210] )
   END_RUNG
   RUNG wire#w1
      Contact( "Unit1.Em7.ControlNodes".jellyRollWinder."step".transition1[210] )
      { S7_Templates := "time_type := Time" } #statTonTime[210].TON(pt := T#1000ms, et =>)
      Move(in := #JOB_2_STEP_20, out1 => "Unit1.Em7.ControlNodes".jellyRollWinder.sequence.status.nextStep)
   END_RUNG
   // the same network as SCL:
   #_w1 := ("Unit1.Em7.ControlNodes".jellyRollWinder.sequence.status.currentStep = #JOB_2_STEP_10) AND "Unit1.Em7.ControlNodes".jellyRollWinder.sequence.status.seqActive;
   "Unit1.Em7.ControlNodes".jellyRollWinder."step".action1[210] := #_w1 AND (NOT "Unit1.Em7.ControlNodes".cm.softCam.jrWinderRearAxisY.clampPos.inPos OR NOT "Unit1.Em7.ControlNodes".cm.softCam.jrWinderFrontAxisY.clampPos.inPos);
   "Unit1.Em7.ControlNodes".jellyRollWinder."step".transition1[210] := #_w1 AND "Unit1.Em7.ControlNodes".cm.softCam.jrWinderRearAxisY.clampPos.inPos AND "Unit1.Em7.ControlNodes".cm.softCam.jrWinderFrontAxisY.clampPos.inPos;
   #statTonTime[210].TON(IN := #_w1 AND "Unit1.Em7.ControlNodes".jellyRollWinder."step".transition1[210],
                         PT := T#1000ms);
   IF #statTonTime[210].Q THEN
       "Unit1.Em7.ControlNodes".jellyRollWinder.sequence.status.nextStep := #JOB_2_STEP_20;
   END_IF;
END_REGION

REGION Network 17: Step[220] : Winder Close
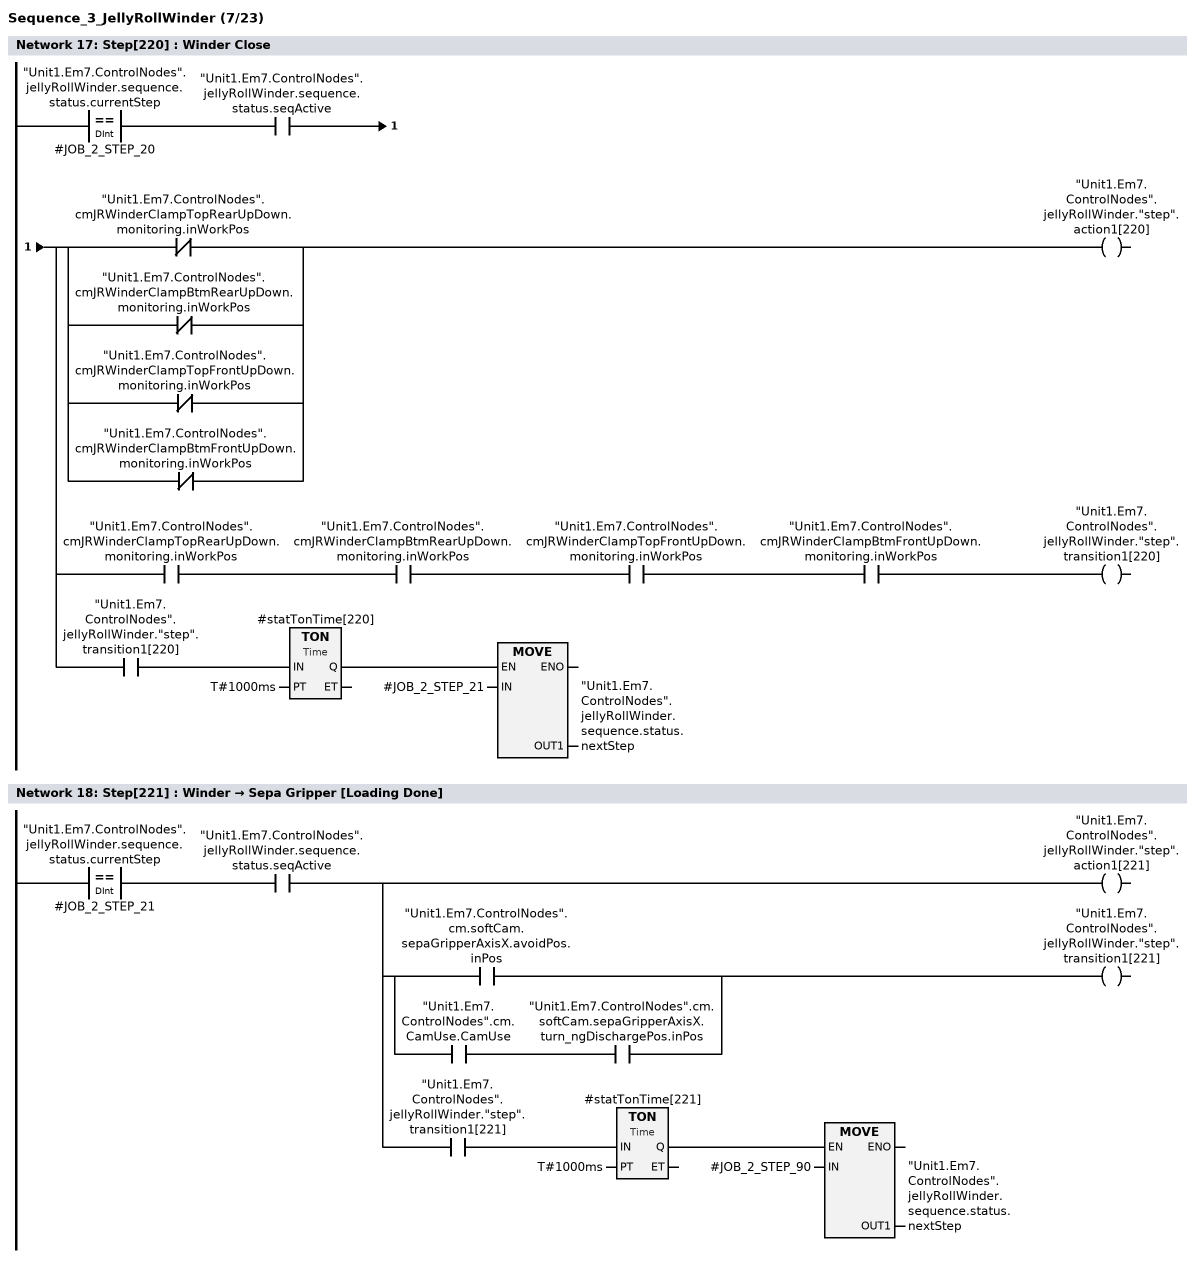
   RUNG wire#powerrail
      { S7_Templates := "SrcType := DInt" } EQ_Contact(in1 := "Unit1.Em7.ControlNodes".jellyRollWinder.sequence.status.currentStep, in2 := #JOB_2_STEP_20)
      Contact( "Unit1.Em7.ControlNodes".jellyRollWinder.sequence.status.seqActive )
      wire#w1
      I_Contact( "Unit1.Em7.ControlNodes".cmJRWinderClampTopRearUpDown.monitoring.inWorkPos )
      wire#w2
      Coil( "Unit1.Em7.ControlNodes".jellyRollWinder."step".action1[220] )
   END_RUNG
   RUNG wire#w1
      I_Contact( "Unit1.Em7.ControlNodes".cmJRWinderClampBtmRearUpDown.monitoring.inWorkPos )
   END_RUNG wire#w2
   RUNG wire#w1
      I_Contact( "Unit1.Em7.ControlNodes".cmJRWinderClampTopFrontUpDown.monitoring.inWorkPos )
   END_RUNG wire#w2
   RUNG wire#w1
      I_Contact( "Unit1.Em7.ControlNodes".cmJRWinderClampBtmFrontUpDown.monitoring.inWorkPos )
   END_RUNG wire#w2
   RUNG wire#w1
      Contact( "Unit1.Em7.ControlNodes".cmJRWinderClampTopRearUpDown.monitoring.inWorkPos )
      Contact( "Unit1.Em7.ControlNodes".cmJRWinderClampBtmRearUpDown.monitoring.inWorkPos )
      Contact( "Unit1.Em7.ControlNodes".cmJRWinderClampTopFrontUpDown.monitoring.inWorkPos )
      Contact( "Unit1.Em7.ControlNodes".cmJRWinderClampBtmFrontUpDown.monitoring.inWorkPos )
      Coil( "Unit1.Em7.ControlNodes".jellyRollWinder."step".transition1[220] )
   END_RUNG
   RUNG wire#w1
      Contact( "Unit1.Em7.ControlNodes".jellyRollWinder."step".transition1[220] )
      { S7_Templates := "time_type := Time" } #statTonTime[220].TON(pt := T#1000ms, et =>)
      Move(in := #JOB_2_STEP_21, out1 => "Unit1.Em7.ControlNodes".jellyRollWinder.sequence.status.nextStep)
   END_RUNG
   // the same network as SCL:
   #_w1 := ("Unit1.Em7.ControlNodes".jellyRollWinder.sequence.status.currentStep = #JOB_2_STEP_20) AND "Unit1.Em7.ControlNodes".jellyRollWinder.sequence.status.seqActive;
   "Unit1.Em7.ControlNodes".jellyRollWinder."step".action1[220] := #_w1 AND (NOT "Unit1.Em7.ControlNodes".cmJRWinderClampTopRearUpDown.monitoring.inWorkPos OR NOT "Unit1.Em7.ControlNodes".cmJRWinderClampBtmRearUpDown.monitoring.inWorkPos OR NOT "Unit1.Em7.ControlNodes".cmJRWinderClampTopFrontUpDown.monitoring.inWorkPos OR NOT "Unit1.Em7.ControlNodes".cmJRWinderClampBtmFrontUpDown.monitoring.inWorkPos);
   "Unit1.Em7.ControlNodes".jellyRollWinder."step".transition1[220] := #_w1 AND "Unit1.Em7.ControlNodes".cmJRWinderClampTopRearUpDown.monitoring.inWorkPos AND "Unit1.Em7.ControlNodes".cmJRWinderClampBtmRearUpDown.monitoring.inWorkPos AND "Unit1.Em7.ControlNodes".cmJRWinderClampTopFrontUpDown.monitoring.inWorkPos AND "Unit1.Em7.ControlNodes".cmJRWinderClampBtmFrontUpDown.monitoring.inWorkPos;
   #statTonTime[220].TON(IN := #_w1 AND "Unit1.Em7.ControlNodes".jellyRollWinder."step".transition1[220],
                         PT := T#1000ms);
   IF #statTonTime[220].Q THEN
       "Unit1.Em7.ControlNodes".jellyRollWinder.sequence.status.nextStep := #JOB_2_STEP_21;
   END_IF;
END_REGION

REGION Network 18: Step[221] : Winder → Sepa Gripper [Loading Done]
   RUNG wire#powerrail
      { S7_Templates := "SrcType := DInt" } EQ_Contact(in1 := "Unit1.Em7.ControlNodes".jellyRollWinder.sequence.status.currentStep, in2 := #JOB_2_STEP_21)
      Contact( "Unit1.Em7.ControlNodes".jellyRollWinder.sequence.status.seqActive )
      wire#w1
      Coil( "Unit1.Em7.ControlNodes".jellyRollWinder."step".action1[221] )
   END_RUNG
   RUNG wire#w1
      Contact( "Unit1.Em7.ControlNodes".cm.softCam.sepaGripperAxisX.avoidPos.inPos )
      wire#w2
      Coil( "Unit1.Em7.ControlNodes".jellyRollWinder."step".transition1[221] )
   END_RUNG
   RUNG wire#w1
      Contact( "Unit1.Em7.ControlNodes".cm.CamUse.CamUse )
      Contact( "Unit1.Em7.ControlNodes".cm.softCam.sepaGripperAxisX.turn_ngDischargePos.inPos )
   END_RUNG wire#w2
   RUNG wire#w1
      Contact( "Unit1.Em7.ControlNodes".jellyRollWinder."step".transition1[221] )
      { S7_Templates := "time_type := Time" } #statTonTime[221].TON(pt := T#1000ms, et =>)
      Move(in := #JOB_2_STEP_90, out1 => "Unit1.Em7.ControlNodes".jellyRollWinder.sequence.status.nextStep)
   END_RUNG
   // the same network as SCL:
   "Unit1.Em7.ControlNodes".jellyRollWinder."step".action1[221] := ("Unit1.Em7.ControlNodes".jellyRollWinder.sequence.status.currentStep = #JOB_2_STEP_21) AND "Unit1.Em7.ControlNodes".jellyRollWinder.sequence.status.seqActive;
   "Unit1.Em7.ControlNodes".jellyRollWinder."step".transition1[221] := ("Unit1.Em7.ControlNodes".jellyRollWinder.sequence.status.currentStep = #JOB_2_STEP_21) AND "Unit1.Em7.ControlNodes".jellyRollWinder.sequence.status.seqActive AND ("Unit1.Em7.ControlNodes".cm.softCam.sepaGripperAxisX.avoidPos.inPos OR ("Unit1.Em7.ControlNodes".cm.CamUse.CamUse AND "Unit1.Em7.ControlNodes".cm.softCam.sepaGripperAxisX.turn_ngDischargePos.inPos));
   #statTonTime[221].TON(IN := ("Unit1.Em7.ControlNodes".jellyRollWinder.sequence.status.currentStep = #JOB_2_STEP_21) AND "Unit1.Em7.ControlNodes".jellyRollWinder.sequence.status.seqActive AND "Unit1.Em7.ControlNodes".jellyRollWinder."step".transition1[221],
                         PT := T#1000ms);
   IF #statTonTime[221].Q THEN
       "Unit1.Em7.ControlNodes".jellyRollWinder.sequence.status.nextStep := #JOB_2_STEP_90;
   END_IF;
END_REGION

REGION Network 19: Step[290] : Job[2] Step End
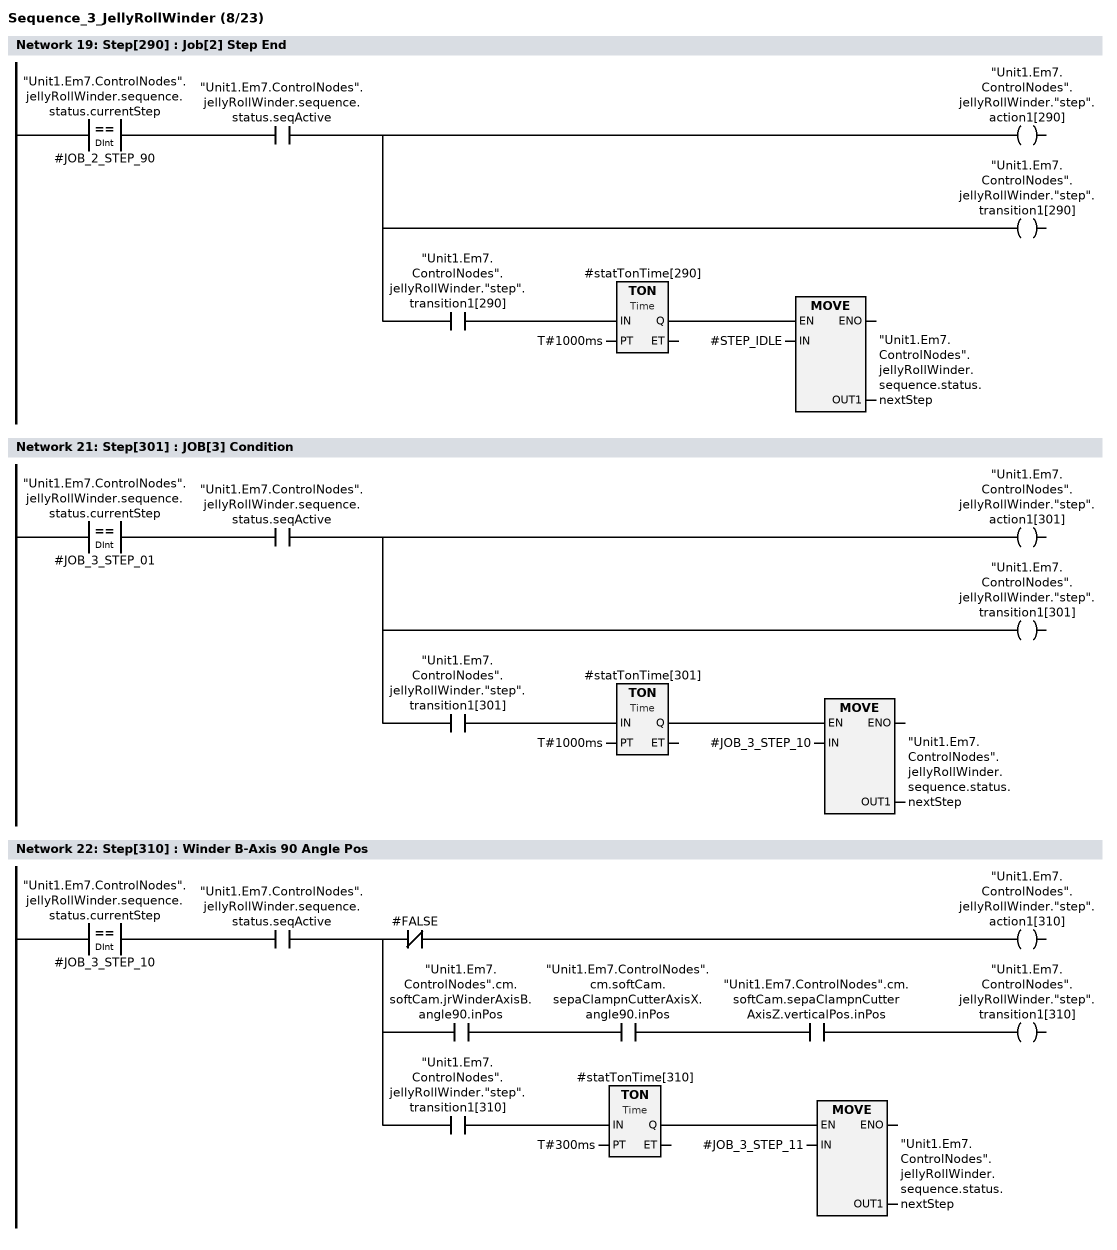
   RUNG wire#powerrail
      { S7_Templates := "SrcType := DInt" } EQ_Contact(in1 := "Unit1.Em7.ControlNodes".jellyRollWinder.sequence.status.currentStep, in2 := #JOB_2_STEP_90)
      Contact( "Unit1.Em7.ControlNodes".jellyRollWinder.sequence.status.seqActive )
      wire#w1
      Coil( "Unit1.Em7.ControlNodes".jellyRollWinder."step".action1[290] )
   END_RUNG
   RUNG wire#w1
      Coil( "Unit1.Em7.ControlNodes".jellyRollWinder."step".transition1[290] )
   END_RUNG
   RUNG wire#w1
      Contact( "Unit1.Em7.ControlNodes".jellyRollWinder."step".transition1[290] )
      { S7_Templates := "time_type := Time" } #statTonTime[290].TON(pt := T#1000ms, et =>)
      Move(in := #STEP_IDLE, out1 => "Unit1.Em7.ControlNodes".jellyRollWinder.sequence.status.nextStep)
   END_RUNG
   // the same network as SCL:
   "Unit1.Em7.ControlNodes".jellyRollWinder."step".action1[290] := ("Unit1.Em7.ControlNodes".jellyRollWinder.sequence.status.currentStep = #JOB_2_STEP_90) AND "Unit1.Em7.ControlNodes".jellyRollWinder.sequence.status.seqActive;
   "Unit1.Em7.ControlNodes".jellyRollWinder."step".transition1[290] := ("Unit1.Em7.ControlNodes".jellyRollWinder.sequence.status.currentStep = #JOB_2_STEP_90) AND "Unit1.Em7.ControlNodes".jellyRollWinder.sequence.status.seqActive;
   #statTonTime[290].TON(IN := ("Unit1.Em7.ControlNodes".jellyRollWinder.sequence.status.currentStep = #JOB_2_STEP_90) AND "Unit1.Em7.ControlNodes".jellyRollWinder.sequence.status.seqActive AND "Unit1.Em7.ControlNodes".jellyRollWinder."step".transition1[290],
                         PT := T#1000ms);
   IF #statTonTime[290].Q THEN
       "Unit1.Em7.ControlNodes".jellyRollWinder.sequence.status.nextStep := #STEP_IDLE;
   END_IF;
END_REGION

REGION Network 20: *************** JOB[3] 1st Winding ************************
END_REGION

REGION Network 21: Step[301] : JOB[3] Condition
   RUNG wire#powerrail
      { S7_Templates := "SrcType := DInt" } EQ_Contact(in1 := "Unit1.Em7.ControlNodes".jellyRollWinder.sequence.status.currentStep, in2 := #JOB_3_STEP_01)
      Contact( "Unit1.Em7.ControlNodes".jellyRollWinder.sequence.status.seqActive )
      wire#w1
      Coil( "Unit1.Em7.ControlNodes".jellyRollWinder."step".action1[301] )
   END_RUNG
   RUNG wire#w1
      Coil( "Unit1.Em7.ControlNodes".jellyRollWinder."step".transition1[301] )
   END_RUNG
   RUNG wire#w1
      Contact( "Unit1.Em7.ControlNodes".jellyRollWinder."step".transition1[301] )
      { S7_Templates := "time_type := Time" } #statTonTime[301].TON(pt := T#1000ms, et =>)
      Move(in := #JOB_3_STEP_10, out1 => "Unit1.Em7.ControlNodes".jellyRollWinder.sequence.status.nextStep)
   END_RUNG
   // the same network as SCL:
   "Unit1.Em7.ControlNodes".jellyRollWinder."step".action1[301] := ("Unit1.Em7.ControlNodes".jellyRollWinder.sequence.status.currentStep = #JOB_3_STEP_01) AND "Unit1.Em7.ControlNodes".jellyRollWinder.sequence.status.seqActive;
   "Unit1.Em7.ControlNodes".jellyRollWinder."step".transition1[301] := ("Unit1.Em7.ControlNodes".jellyRollWinder.sequence.status.currentStep = #JOB_3_STEP_01) AND "Unit1.Em7.ControlNodes".jellyRollWinder.sequence.status.seqActive;
   #statTonTime[301].TON(IN := ("Unit1.Em7.ControlNodes".jellyRollWinder.sequence.status.currentStep = #JOB_3_STEP_01) AND "Unit1.Em7.ControlNodes".jellyRollWinder.sequence.status.seqActive AND "Unit1.Em7.ControlNodes".jellyRollWinder."step".transition1[301],
                         PT := T#1000ms);
   IF #statTonTime[301].Q THEN
       "Unit1.Em7.ControlNodes".jellyRollWinder.sequence.status.nextStep := #JOB_3_STEP_10;
   END_IF;
END_REGION

REGION Network 22: Step[310] : Winder B-Axis 90 Angle Pos
   RUNG wire#powerrail
      { S7_Templates := "SrcType := DInt" } EQ_Contact(in1 := "Unit1.Em7.ControlNodes".jellyRollWinder.sequence.status.currentStep, in2 := #JOB_3_STEP_10)
      Contact( "Unit1.Em7.ControlNodes".jellyRollWinder.sequence.status.seqActive )
      wire#w1
      I_Contact( #FALSE )
      Coil( "Unit1.Em7.ControlNodes".jellyRollWinder."step".action1[310] )
   END_RUNG
   RUNG wire#w1
      Contact( "Unit1.Em7.ControlNodes".cm.softCam.jrWinderAxisB.angle90.inPos )
      Contact( "Unit1.Em7.ControlNodes".cm.softCam.sepaClampnCutterAxisX.angle90.inPos )
      Contact( "Unit1.Em7.ControlNodes".cm.softCam.sepaClampnCutterAxisZ.verticalPos.inPos )
      Coil( "Unit1.Em7.ControlNodes".jellyRollWinder."step".transition1[310] )
   END_RUNG
   RUNG wire#w1
      Contact( "Unit1.Em7.ControlNodes".jellyRollWinder."step".transition1[310] )
      { S7_Templates := "time_type := Time" } #statTonTime[310].TON(pt := T#300ms, et =>)
      Move(in := #JOB_3_STEP_11, out1 => "Unit1.Em7.ControlNodes".jellyRollWinder.sequence.status.nextStep)
   END_RUNG
   // the same network as SCL:
   #_w1 := ("Unit1.Em7.ControlNodes".jellyRollWinder.sequence.status.currentStep = #JOB_3_STEP_10) AND "Unit1.Em7.ControlNodes".jellyRollWinder.sequence.status.seqActive;
   "Unit1.Em7.ControlNodes".jellyRollWinder."step".action1[310] := #_w1 AND NOT #FALSE;
   "Unit1.Em7.ControlNodes".jellyRollWinder."step".transition1[310] := #_w1 AND "Unit1.Em7.ControlNodes".cm.softCam.jrWinderAxisB.angle90.inPos AND "Unit1.Em7.ControlNodes".cm.softCam.sepaClampnCutterAxisX.angle90.inPos AND "Unit1.Em7.ControlNodes".cm.softCam.sepaClampnCutterAxisZ.verticalPos.inPos;
   #statTonTime[310].TON(IN := #_w1 AND "Unit1.Em7.ControlNodes".jellyRollWinder."step".transition1[310],
                         PT := T#300ms);
   IF #statTonTime[310].Q THEN
       "Unit1.Em7.ControlNodes".jellyRollWinder.sequence.status.nextStep := #JOB_3_STEP_11;
   END_IF;
END_REGION

REGION Network 23: Step[311] : Winder B-Axis 180 Angle Pos
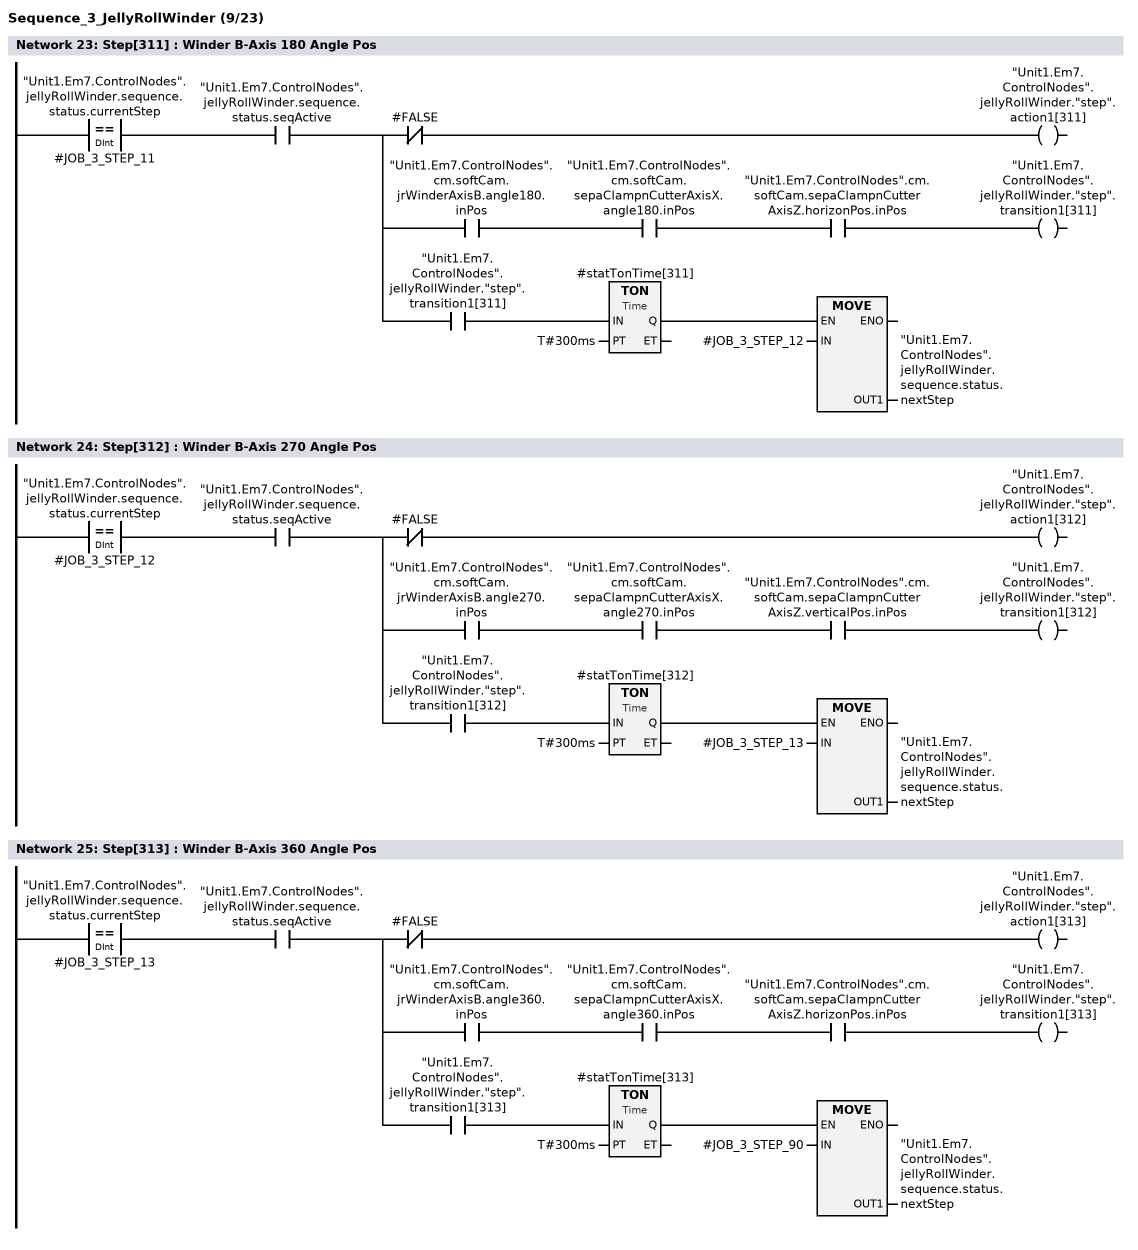
   RUNG wire#powerrail
      { S7_Templates := "SrcType := DInt" } EQ_Contact(in1 := "Unit1.Em7.ControlNodes".jellyRollWinder.sequence.status.currentStep, in2 := #JOB_3_STEP_11)
      Contact( "Unit1.Em7.ControlNodes".jellyRollWinder.sequence.status.seqActive )
      wire#w1
      I_Contact( #FALSE )
      Coil( "Unit1.Em7.ControlNodes".jellyRollWinder."step".action1[311] )
   END_RUNG
   RUNG wire#w1
      Contact( "Unit1.Em7.ControlNodes".cm.softCam.jrWinderAxisB.angle180.inPos )
      Contact( "Unit1.Em7.ControlNodes".cm.softCam.sepaClampnCutterAxisX.angle180.inPos )
      Contact( "Unit1.Em7.ControlNodes".cm.softCam.sepaClampnCutterAxisZ.horizonPos.inPos )
      Coil( "Unit1.Em7.ControlNodes".jellyRollWinder."step".transition1[311] )
   END_RUNG
   RUNG wire#w1
      Contact( "Unit1.Em7.ControlNodes".jellyRollWinder."step".transition1[311] )
      { S7_Templates := "time_type := Time" } #statTonTime[311].TON(pt := T#300ms, et =>)
      Move(in := #JOB_3_STEP_12, out1 => "Unit1.Em7.ControlNodes".jellyRollWinder.sequence.status.nextStep)
   END_RUNG
   // the same network as SCL:
   #_w1 := ("Unit1.Em7.ControlNodes".jellyRollWinder.sequence.status.currentStep = #JOB_3_STEP_11) AND "Unit1.Em7.ControlNodes".jellyRollWinder.sequence.status.seqActive;
   "Unit1.Em7.ControlNodes".jellyRollWinder."step".action1[311] := #_w1 AND NOT #FALSE;
   "Unit1.Em7.ControlNodes".jellyRollWinder."step".transition1[311] := #_w1 AND "Unit1.Em7.ControlNodes".cm.softCam.jrWinderAxisB.angle180.inPos AND "Unit1.Em7.ControlNodes".cm.softCam.sepaClampnCutterAxisX.angle180.inPos AND "Unit1.Em7.ControlNodes".cm.softCam.sepaClampnCutterAxisZ.horizonPos.inPos;
   #statTonTime[311].TON(IN := #_w1 AND "Unit1.Em7.ControlNodes".jellyRollWinder."step".transition1[311],
                         PT := T#300ms);
   IF #statTonTime[311].Q THEN
       "Unit1.Em7.ControlNodes".jellyRollWinder.sequence.status.nextStep := #JOB_3_STEP_12;
   END_IF;
END_REGION

REGION Network 24: Step[312] : Winder B-Axis 270 Angle Pos
   RUNG wire#powerrail
      { S7_Templates := "SrcType := DInt" } EQ_Contact(in1 := "Unit1.Em7.ControlNodes".jellyRollWinder.sequence.status.currentStep, in2 := #JOB_3_STEP_12)
      Contact( "Unit1.Em7.ControlNodes".jellyRollWinder.sequence.status.seqActive )
      wire#w1
      I_Contact( #FALSE )
      Coil( "Unit1.Em7.ControlNodes".jellyRollWinder."step".action1[312] )
   END_RUNG
   RUNG wire#w1
      Contact( "Unit1.Em7.ControlNodes".cm.softCam.jrWinderAxisB.angle270.inPos )
      Contact( "Unit1.Em7.ControlNodes".cm.softCam.sepaClampnCutterAxisX.angle270.inPos )
      Contact( "Unit1.Em7.ControlNodes".cm.softCam.sepaClampnCutterAxisZ.verticalPos.inPos )
      Coil( "Unit1.Em7.ControlNodes".jellyRollWinder."step".transition1[312] )
   END_RUNG
   RUNG wire#w1
      Contact( "Unit1.Em7.ControlNodes".jellyRollWinder."step".transition1[312] )
      { S7_Templates := "time_type := Time" } #statTonTime[312].TON(pt := T#300ms, et =>)
      Move(in := #JOB_3_STEP_13, out1 => "Unit1.Em7.ControlNodes".jellyRollWinder.sequence.status.nextStep)
   END_RUNG
   // the same network as SCL:
   #_w1 := ("Unit1.Em7.ControlNodes".jellyRollWinder.sequence.status.currentStep = #JOB_3_STEP_12) AND "Unit1.Em7.ControlNodes".jellyRollWinder.sequence.status.seqActive;
   "Unit1.Em7.ControlNodes".jellyRollWinder."step".action1[312] := #_w1 AND NOT #FALSE;
   "Unit1.Em7.ControlNodes".jellyRollWinder."step".transition1[312] := #_w1 AND "Unit1.Em7.ControlNodes".cm.softCam.jrWinderAxisB.angle270.inPos AND "Unit1.Em7.ControlNodes".cm.softCam.sepaClampnCutterAxisX.angle270.inPos AND "Unit1.Em7.ControlNodes".cm.softCam.sepaClampnCutterAxisZ.verticalPos.inPos;
   #statTonTime[312].TON(IN := #_w1 AND "Unit1.Em7.ControlNodes".jellyRollWinder."step".transition1[312],
                         PT := T#300ms);
   IF #statTonTime[312].Q THEN
       "Unit1.Em7.ControlNodes".jellyRollWinder.sequence.status.nextStep := #JOB_3_STEP_13;
   END_IF;
END_REGION

REGION Network 25: Step[313] : Winder B-Axis 360 Angle Pos
   RUNG wire#powerrail
      { S7_Templates := "SrcType := DInt" } EQ_Contact(in1 := "Unit1.Em7.ControlNodes".jellyRollWinder.sequence.status.currentStep, in2 := #JOB_3_STEP_13)
      Contact( "Unit1.Em7.ControlNodes".jellyRollWinder.sequence.status.seqActive )
      wire#w1
      I_Contact( #FALSE )
      Coil( "Unit1.Em7.ControlNodes".jellyRollWinder."step".action1[313] )
   END_RUNG
   RUNG wire#w1
      Contact( "Unit1.Em7.ControlNodes".cm.softCam.jrWinderAxisB.angle360.inPos )
      Contact( "Unit1.Em7.ControlNodes".cm.softCam.sepaClampnCutterAxisX.angle360.inPos )
      Contact( "Unit1.Em7.ControlNodes".cm.softCam.sepaClampnCutterAxisZ.horizonPos.inPos )
      Coil( "Unit1.Em7.ControlNodes".jellyRollWinder."step".transition1[313] )
   END_RUNG
   RUNG wire#w1
      Contact( "Unit1.Em7.ControlNodes".jellyRollWinder."step".transition1[313] )
      { S7_Templates := "time_type := Time" } #statTonTime[313].TON(pt := T#300ms, et =>)
      Move(in := #JOB_3_STEP_90, out1 => "Unit1.Em7.ControlNodes".jellyRollWinder.sequence.status.nextStep)
   END_RUNG
   // the same network as SCL:
   #_w1 := ("Unit1.Em7.ControlNodes".jellyRollWinder.sequence.status.currentStep = #JOB_3_STEP_13) AND "Unit1.Em7.ControlNodes".jellyRollWinder.sequence.status.seqActive;
   "Unit1.Em7.ControlNodes".jellyRollWinder."step".action1[313] := #_w1 AND NOT #FALSE;
   "Unit1.Em7.ControlNodes".jellyRollWinder."step".transition1[313] := #_w1 AND "Unit1.Em7.ControlNodes".cm.softCam.jrWinderAxisB.angle360.inPos AND "Unit1.Em7.ControlNodes".cm.softCam.sepaClampnCutterAxisX.angle360.inPos AND "Unit1.Em7.ControlNodes".cm.softCam.sepaClampnCutterAxisZ.horizonPos.inPos;
   #statTonTime[313].TON(IN := #_w1 AND "Unit1.Em7.ControlNodes".jellyRollWinder."step".transition1[313],
                         PT := T#300ms);
   IF #statTonTime[313].Q THEN
       "Unit1.Em7.ControlNodes".jellyRollWinder.sequence.status.nextStep := #JOB_3_STEP_90;
   END_IF;
END_REGION

REGION Network 26: Step[390] : Job[3] Step End
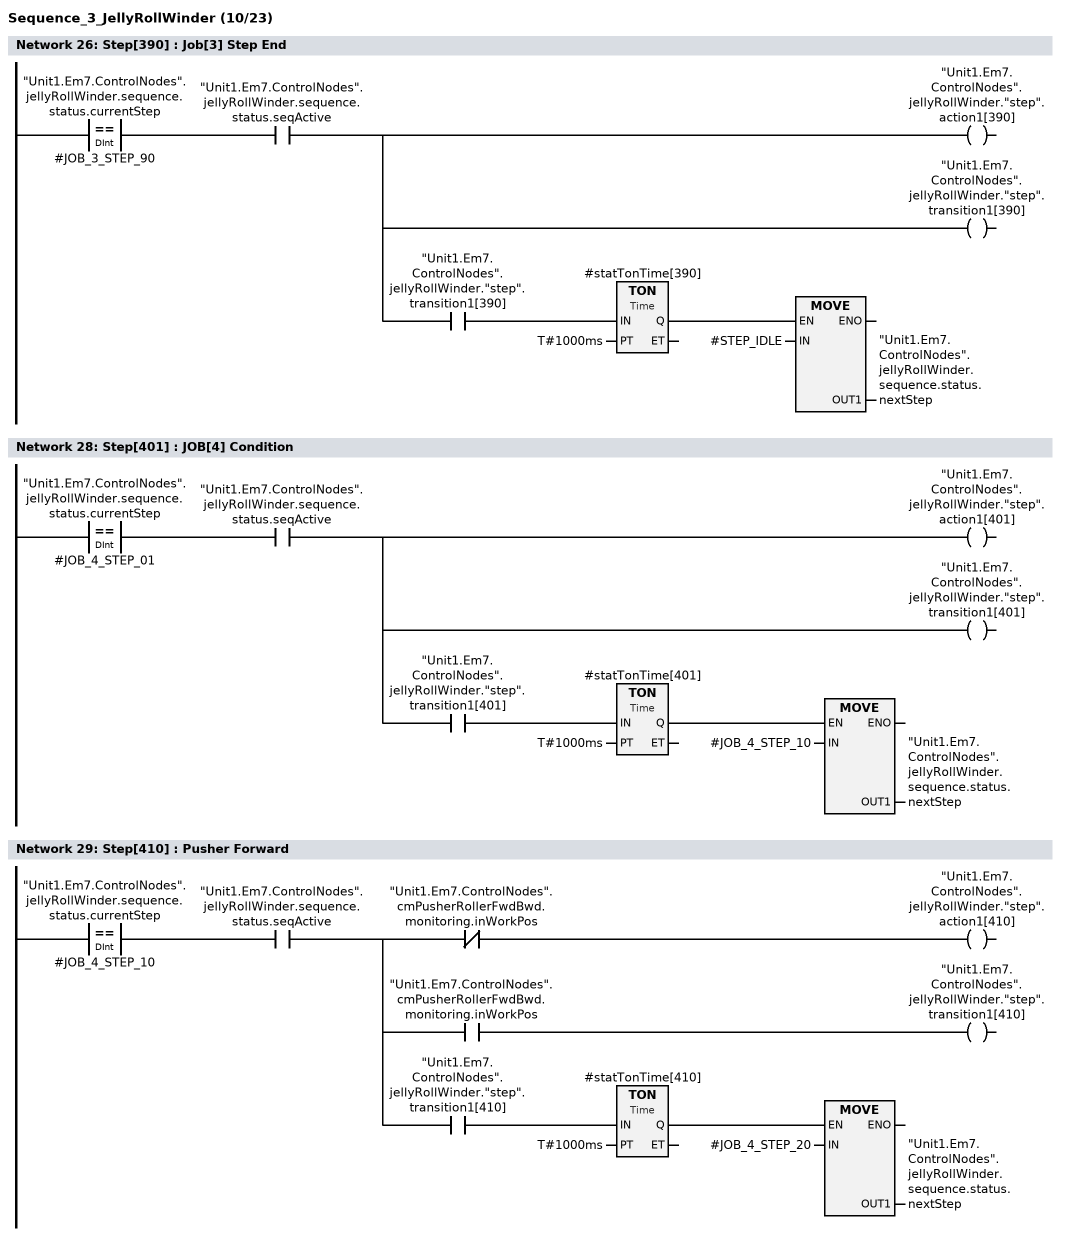
   RUNG wire#powerrail
      { S7_Templates := "SrcType := DInt" } EQ_Contact(in1 := "Unit1.Em7.ControlNodes".jellyRollWinder.sequence.status.currentStep, in2 := #JOB_3_STEP_90)
      Contact( "Unit1.Em7.ControlNodes".jellyRollWinder.sequence.status.seqActive )
      wire#w1
      Coil( "Unit1.Em7.ControlNodes".jellyRollWinder."step".action1[390] )
   END_RUNG
   RUNG wire#w1
      Coil( "Unit1.Em7.ControlNodes".jellyRollWinder."step".transition1[390] )
   END_RUNG
   RUNG wire#w1
      Contact( "Unit1.Em7.ControlNodes".jellyRollWinder."step".transition1[390] )
      { S7_Templates := "time_type := Time" } #statTonTime[390].TON(pt := T#1000ms, et =>)
      Move(in := #STEP_IDLE, out1 => "Unit1.Em7.ControlNodes".jellyRollWinder.sequence.status.nextStep)
   END_RUNG
   // the same network as SCL:
   "Unit1.Em7.ControlNodes".jellyRollWinder."step".action1[390] := ("Unit1.Em7.ControlNodes".jellyRollWinder.sequence.status.currentStep = #JOB_3_STEP_90) AND "Unit1.Em7.ControlNodes".jellyRollWinder.sequence.status.seqActive;
   "Unit1.Em7.ControlNodes".jellyRollWinder."step".transition1[390] := ("Unit1.Em7.ControlNodes".jellyRollWinder.sequence.status.currentStep = #JOB_3_STEP_90) AND "Unit1.Em7.ControlNodes".jellyRollWinder.sequence.status.seqActive;
   #statTonTime[390].TON(IN := ("Unit1.Em7.ControlNodes".jellyRollWinder.sequence.status.currentStep = #JOB_3_STEP_90) AND "Unit1.Em7.ControlNodes".jellyRollWinder.sequence.status.seqActive AND "Unit1.Em7.ControlNodes".jellyRollWinder."step".transition1[390],
                         PT := T#1000ms);
   IF #statTonTime[390].Q THEN
       "Unit1.Em7.ControlNodes".jellyRollWinder.sequence.status.nextStep := #STEP_IDLE;
   END_IF;
END_REGION

REGION Network 27: *************** JOB[4] Pusher Ready ************************
END_REGION

REGION Network 28: Step[401] : JOB[4] Condition
   RUNG wire#powerrail
      { S7_Templates := "SrcType := DInt" } EQ_Contact(in1 := "Unit1.Em7.ControlNodes".jellyRollWinder.sequence.status.currentStep, in2 := #JOB_4_STEP_01)
      Contact( "Unit1.Em7.ControlNodes".jellyRollWinder.sequence.status.seqActive )
      wire#w1
      Coil( "Unit1.Em7.ControlNodes".jellyRollWinder."step".action1[401] )
   END_RUNG
   RUNG wire#w1
      Coil( "Unit1.Em7.ControlNodes".jellyRollWinder."step".transition1[401] )
   END_RUNG
   RUNG wire#w1
      Contact( "Unit1.Em7.ControlNodes".jellyRollWinder."step".transition1[401] )
      { S7_Templates := "time_type := Time" } #statTonTime[401].TON(pt := T#1000ms, et =>)
      Move(in := #JOB_4_STEP_10, out1 => "Unit1.Em7.ControlNodes".jellyRollWinder.sequence.status.nextStep)
   END_RUNG
   // the same network as SCL:
   "Unit1.Em7.ControlNodes".jellyRollWinder."step".action1[401] := ("Unit1.Em7.ControlNodes".jellyRollWinder.sequence.status.currentStep = #JOB_4_STEP_01) AND "Unit1.Em7.ControlNodes".jellyRollWinder.sequence.status.seqActive;
   "Unit1.Em7.ControlNodes".jellyRollWinder."step".transition1[401] := ("Unit1.Em7.ControlNodes".jellyRollWinder.sequence.status.currentStep = #JOB_4_STEP_01) AND "Unit1.Em7.ControlNodes".jellyRollWinder.sequence.status.seqActive;
   #statTonTime[401].TON(IN := ("Unit1.Em7.ControlNodes".jellyRollWinder.sequence.status.currentStep = #JOB_4_STEP_01) AND "Unit1.Em7.ControlNodes".jellyRollWinder.sequence.status.seqActive AND "Unit1.Em7.ControlNodes".jellyRollWinder."step".transition1[401],
                         PT := T#1000ms);
   IF #statTonTime[401].Q THEN
       "Unit1.Em7.ControlNodes".jellyRollWinder.sequence.status.nextStep := #JOB_4_STEP_10;
   END_IF;
END_REGION

REGION Network 29: Step[410] : Pusher Forward
   RUNG wire#powerrail
      { S7_Templates := "SrcType := DInt" } EQ_Contact(in1 := "Unit1.Em7.ControlNodes".jellyRollWinder.sequence.status.currentStep, in2 := #JOB_4_STEP_10)
      Contact( "Unit1.Em7.ControlNodes".jellyRollWinder.sequence.status.seqActive )
      wire#w1
      I_Contact( "Unit1.Em7.ControlNodes".cmPusherRollerFwdBwd.monitoring.inWorkPos )
      Coil( "Unit1.Em7.ControlNodes".jellyRollWinder."step".action1[410] )
   END_RUNG
   RUNG wire#w1
      Contact( "Unit1.Em7.ControlNodes".cmPusherRollerFwdBwd.monitoring.inWorkPos )
      Coil( "Unit1.Em7.ControlNodes".jellyRollWinder."step".transition1[410] )
   END_RUNG
   RUNG wire#w1
      Contact( "Unit1.Em7.ControlNodes".jellyRollWinder."step".transition1[410] )
      { S7_Templates := "time_type := Time" } #statTonTime[410].TON(pt := T#1000ms, et =>)
      Move(in := #JOB_4_STEP_20, out1 => "Unit1.Em7.ControlNodes".jellyRollWinder.sequence.status.nextStep)
   END_RUNG
   // the same network as SCL:
   #_w1 := ("Unit1.Em7.ControlNodes".jellyRollWinder.sequence.status.currentStep = #JOB_4_STEP_10) AND "Unit1.Em7.ControlNodes".jellyRollWinder.sequence.status.seqActive;
   "Unit1.Em7.ControlNodes".jellyRollWinder."step".action1[410] := #_w1 AND NOT "Unit1.Em7.ControlNodes".cmPusherRollerFwdBwd.monitoring.inWorkPos;
   "Unit1.Em7.ControlNodes".jellyRollWinder."step".transition1[410] := #_w1 AND "Unit1.Em7.ControlNodes".cmPusherRollerFwdBwd.monitoring.inWorkPos;
   #statTonTime[410].TON(IN := #_w1 AND "Unit1.Em7.ControlNodes".jellyRollWinder."step".transition1[410],
                         PT := T#1000ms);
   IF #statTonTime[410].Q THEN
       "Unit1.Em7.ControlNodes".jellyRollWinder.sequence.status.nextStep := #JOB_4_STEP_20;
   END_IF;
END_REGION

REGION Network 30: Step[420] : Pusher Z-Axis Work(=Down) Pos
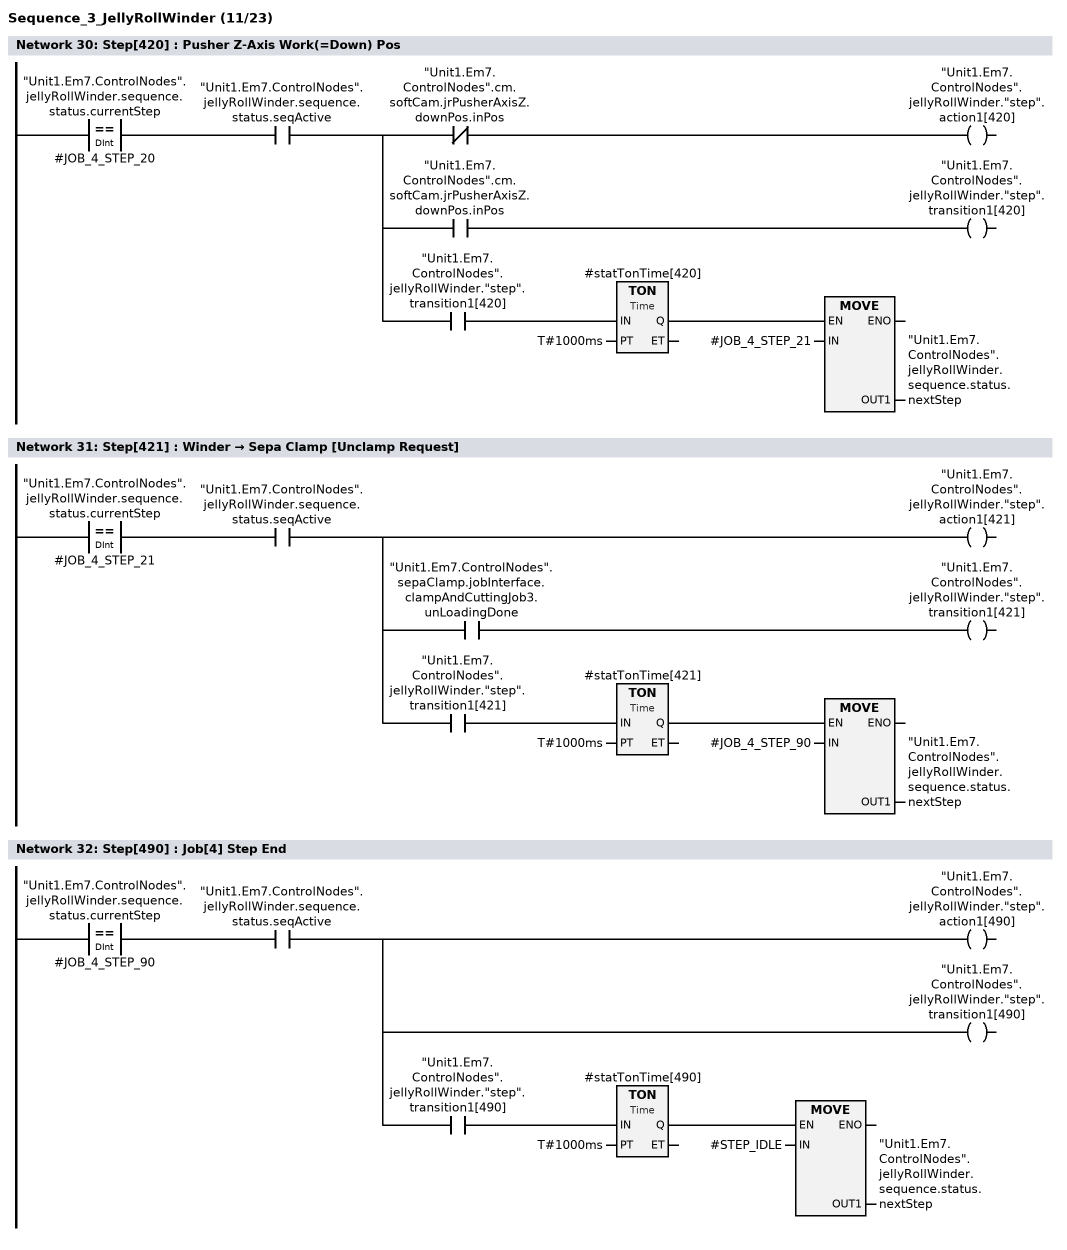
   RUNG wire#powerrail
      { S7_Templates := "SrcType := DInt" } EQ_Contact(in1 := "Unit1.Em7.ControlNodes".jellyRollWinder.sequence.status.currentStep, in2 := #JOB_4_STEP_20)
      Contact( "Unit1.Em7.ControlNodes".jellyRollWinder.sequence.status.seqActive )
      wire#w1
      I_Contact( "Unit1.Em7.ControlNodes".cm.softCam.jrPusherAxisZ.downPos.inPos )
      Coil( "Unit1.Em7.ControlNodes".jellyRollWinder."step".action1[420] )
   END_RUNG
   RUNG wire#w1
      Contact( "Unit1.Em7.ControlNodes".cm.softCam.jrPusherAxisZ.downPos.inPos )
      Coil( "Unit1.Em7.ControlNodes".jellyRollWinder."step".transition1[420] )
   END_RUNG
   RUNG wire#w1
      Contact( "Unit1.Em7.ControlNodes".jellyRollWinder."step".transition1[420] )
      { S7_Templates := "time_type := Time" } #statTonTime[420].TON(pt := T#1000ms, et =>)
      Move(in := #JOB_4_STEP_21, out1 => "Unit1.Em7.ControlNodes".jellyRollWinder.sequence.status.nextStep)
   END_RUNG
   // the same network as SCL:
   #_w1 := ("Unit1.Em7.ControlNodes".jellyRollWinder.sequence.status.currentStep = #JOB_4_STEP_20) AND "Unit1.Em7.ControlNodes".jellyRollWinder.sequence.status.seqActive;
   "Unit1.Em7.ControlNodes".jellyRollWinder."step".action1[420] := #_w1 AND NOT "Unit1.Em7.ControlNodes".cm.softCam.jrPusherAxisZ.downPos.inPos;
   "Unit1.Em7.ControlNodes".jellyRollWinder."step".transition1[420] := #_w1 AND "Unit1.Em7.ControlNodes".cm.softCam.jrPusherAxisZ.downPos.inPos;
   #statTonTime[420].TON(IN := #_w1 AND "Unit1.Em7.ControlNodes".jellyRollWinder."step".transition1[420],
                         PT := T#1000ms);
   IF #statTonTime[420].Q THEN
       "Unit1.Em7.ControlNodes".jellyRollWinder.sequence.status.nextStep := #JOB_4_STEP_21;
   END_IF;
END_REGION

REGION Network 31: Step[421] : Winder → Sepa Clamp [Unclamp Request]
   RUNG wire#powerrail
      { S7_Templates := "SrcType := DInt" } EQ_Contact(in1 := "Unit1.Em7.ControlNodes".jellyRollWinder.sequence.status.currentStep, in2 := #JOB_4_STEP_21)
      Contact( "Unit1.Em7.ControlNodes".jellyRollWinder.sequence.status.seqActive )
      wire#w1
      Coil( "Unit1.Em7.ControlNodes".jellyRollWinder."step".action1[421] )
   END_RUNG
   RUNG wire#w1
      Contact( "Unit1.Em7.ControlNodes".sepaClamp.jobInterface.clampAndCuttingJob3.unLoadingDone )
      Coil( "Unit1.Em7.ControlNodes".jellyRollWinder."step".transition1[421] )
   END_RUNG
   RUNG wire#w1
      Contact( "Unit1.Em7.ControlNodes".jellyRollWinder."step".transition1[421] )
      { S7_Templates := "time_type := Time" } #statTonTime[421].TON(pt := T#1000ms, et =>)
      Move(in := #JOB_4_STEP_90, out1 => "Unit1.Em7.ControlNodes".jellyRollWinder.sequence.status.nextStep)
   END_RUNG
   // the same network as SCL:
   "Unit1.Em7.ControlNodes".jellyRollWinder."step".action1[421] := ("Unit1.Em7.ControlNodes".jellyRollWinder.sequence.status.currentStep = #JOB_4_STEP_21) AND "Unit1.Em7.ControlNodes".jellyRollWinder.sequence.status.seqActive;
   "Unit1.Em7.ControlNodes".jellyRollWinder."step".transition1[421] := ("Unit1.Em7.ControlNodes".jellyRollWinder.sequence.status.currentStep = #JOB_4_STEP_21) AND "Unit1.Em7.ControlNodes".jellyRollWinder.sequence.status.seqActive AND "Unit1.Em7.ControlNodes".sepaClamp.jobInterface.clampAndCuttingJob3.unLoadingDone;
   #statTonTime[421].TON(IN := ("Unit1.Em7.ControlNodes".jellyRollWinder.sequence.status.currentStep = #JOB_4_STEP_21) AND "Unit1.Em7.ControlNodes".jellyRollWinder.sequence.status.seqActive AND "Unit1.Em7.ControlNodes".jellyRollWinder."step".transition1[421],
                         PT := T#1000ms);
   IF #statTonTime[421].Q THEN
       "Unit1.Em7.ControlNodes".jellyRollWinder.sequence.status.nextStep := #JOB_4_STEP_90;
   END_IF;
END_REGION

REGION Network 32: Step[490] : Job[4] Step End
   RUNG wire#powerrail
      { S7_Templates := "SrcType := DInt" } EQ_Contact(in1 := "Unit1.Em7.ControlNodes".jellyRollWinder.sequence.status.currentStep, in2 := #JOB_4_STEP_90)
      Contact( "Unit1.Em7.ControlNodes".jellyRollWinder.sequence.status.seqActive )
      wire#w1
      Coil( "Unit1.Em7.ControlNodes".jellyRollWinder."step".action1[490] )
   END_RUNG
   RUNG wire#w1
      Coil( "Unit1.Em7.ControlNodes".jellyRollWinder."step".transition1[490] )
   END_RUNG
   RUNG wire#w1
      Contact( "Unit1.Em7.ControlNodes".jellyRollWinder."step".transition1[490] )
      { S7_Templates := "time_type := Time" } #statTonTime[490].TON(pt := T#1000ms, et =>)
      Move(in := #STEP_IDLE, out1 => "Unit1.Em7.ControlNodes".jellyRollWinder.sequence.status.nextStep)
   END_RUNG
   // the same network as SCL:
   "Unit1.Em7.ControlNodes".jellyRollWinder."step".action1[490] := ("Unit1.Em7.ControlNodes".jellyRollWinder.sequence.status.currentStep = #JOB_4_STEP_90) AND "Unit1.Em7.ControlNodes".jellyRollWinder.sequence.status.seqActive;
   "Unit1.Em7.ControlNodes".jellyRollWinder."step".transition1[490] := ("Unit1.Em7.ControlNodes".jellyRollWinder.sequence.status.currentStep = #JOB_4_STEP_90) AND "Unit1.Em7.ControlNodes".jellyRollWinder.sequence.status.seqActive;
   #statTonTime[490].TON(IN := ("Unit1.Em7.ControlNodes".jellyRollWinder.sequence.status.currentStep = #JOB_4_STEP_90) AND "Unit1.Em7.ControlNodes".jellyRollWinder.sequence.status.seqActive AND "Unit1.Em7.ControlNodes".jellyRollWinder."step".transition1[490],
                         PT := T#1000ms);
   IF #statTonTime[490].Q THEN
       "Unit1.Em7.ControlNodes".jellyRollWinder.sequence.status.nextStep := #STEP_IDLE;
   END_IF;
END_REGION

REGION Network 33: *************** JOB[5] 2nd Winding ************************
END_REGION

REGION Network 34: Step[501] : JOB[5] Condition
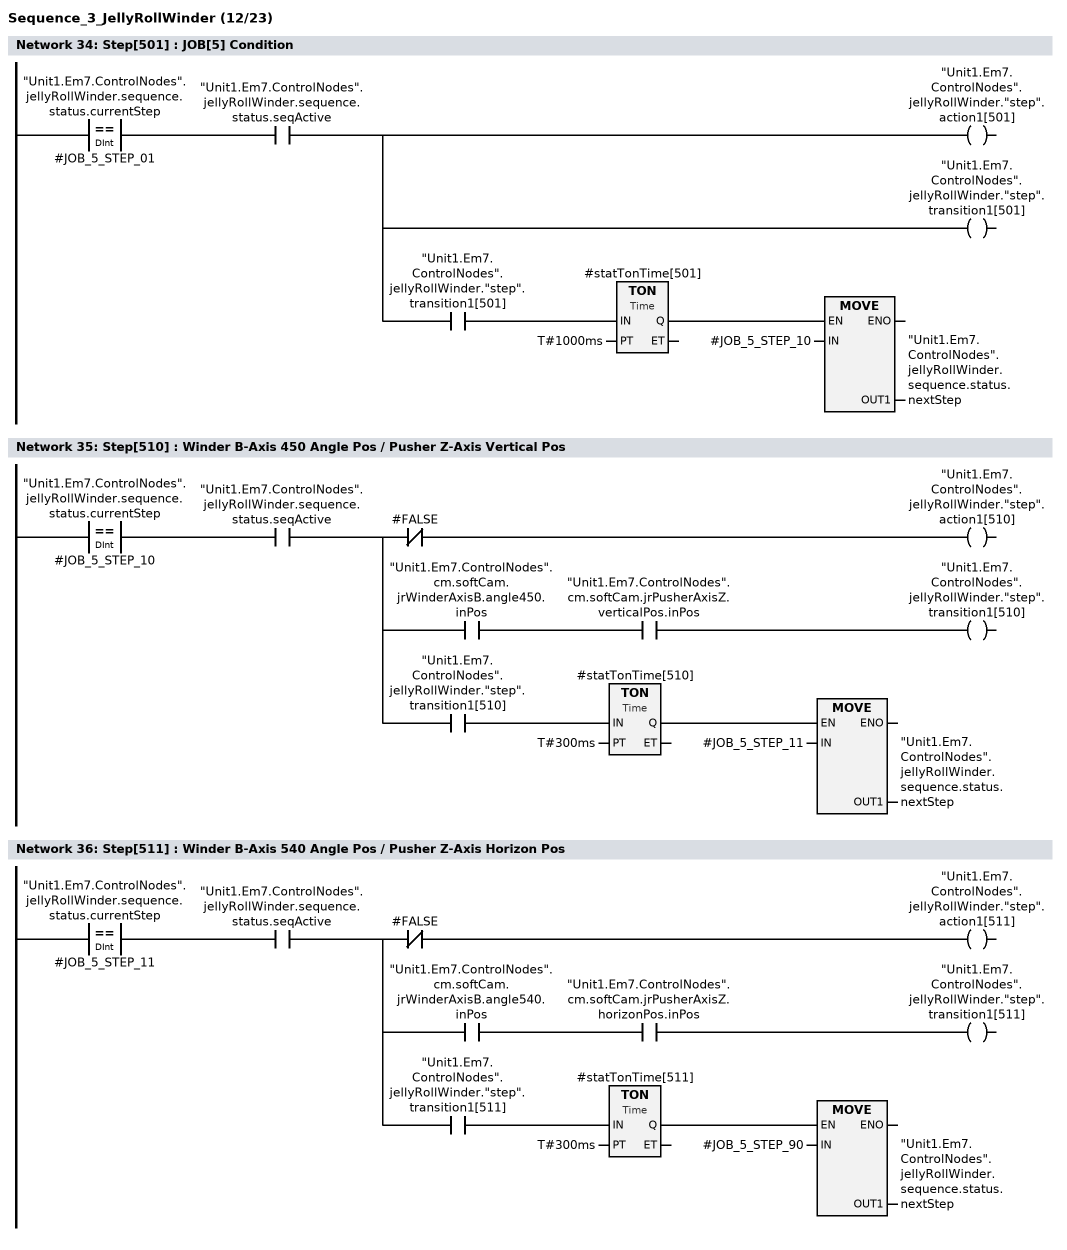
   RUNG wire#powerrail
      { S7_Templates := "SrcType := DInt" } EQ_Contact(in1 := "Unit1.Em7.ControlNodes".jellyRollWinder.sequence.status.currentStep, in2 := #JOB_5_STEP_01)
      Contact( "Unit1.Em7.ControlNodes".jellyRollWinder.sequence.status.seqActive )
      wire#w1
      Coil( "Unit1.Em7.ControlNodes".jellyRollWinder."step".action1[501] )
   END_RUNG
   RUNG wire#w1
      Coil( "Unit1.Em7.ControlNodes".jellyRollWinder."step".transition1[501] )
   END_RUNG
   RUNG wire#w1
      Contact( "Unit1.Em7.ControlNodes".jellyRollWinder."step".transition1[501] )
      { S7_Templates := "time_type := Time" } #statTonTime[501].TON(pt := T#1000ms, et =>)
      Move(in := #JOB_5_STEP_10, out1 => "Unit1.Em7.ControlNodes".jellyRollWinder.sequence.status.nextStep)
   END_RUNG
   // the same network as SCL:
   "Unit1.Em7.ControlNodes".jellyRollWinder."step".action1[501] := ("Unit1.Em7.ControlNodes".jellyRollWinder.sequence.status.currentStep = #JOB_5_STEP_01) AND "Unit1.Em7.ControlNodes".jellyRollWinder.sequence.status.seqActive;
   "Unit1.Em7.ControlNodes".jellyRollWinder."step".transition1[501] := ("Unit1.Em7.ControlNodes".jellyRollWinder.sequence.status.currentStep = #JOB_5_STEP_01) AND "Unit1.Em7.ControlNodes".jellyRollWinder.sequence.status.seqActive;
   #statTonTime[501].TON(IN := ("Unit1.Em7.ControlNodes".jellyRollWinder.sequence.status.currentStep = #JOB_5_STEP_01) AND "Unit1.Em7.ControlNodes".jellyRollWinder.sequence.status.seqActive AND "Unit1.Em7.ControlNodes".jellyRollWinder."step".transition1[501],
                         PT := T#1000ms);
   IF #statTonTime[501].Q THEN
       "Unit1.Em7.ControlNodes".jellyRollWinder.sequence.status.nextStep := #JOB_5_STEP_10;
   END_IF;
END_REGION

REGION Network 35: Step[510] : Winder B-Axis 450 Angle Pos / Pusher Z-Axis Vertical Pos
   RUNG wire#powerrail
      { S7_Templates := "SrcType := DInt" } EQ_Contact(in1 := "Unit1.Em7.ControlNodes".jellyRollWinder.sequence.status.currentStep, in2 := #JOB_5_STEP_10)
      Contact( "Unit1.Em7.ControlNodes".jellyRollWinder.sequence.status.seqActive )
      wire#w1
      I_Contact( #FALSE )
      Coil( "Unit1.Em7.ControlNodes".jellyRollWinder."step".action1[510] )
   END_RUNG
   RUNG wire#w1
      Contact( "Unit1.Em7.ControlNodes".cm.softCam.jrWinderAxisB.angle450.inPos )
      Contact( "Unit1.Em7.ControlNodes".cm.softCam.jrPusherAxisZ.verticalPos.inPos )
      Coil( "Unit1.Em7.ControlNodes".jellyRollWinder."step".transition1[510] )
   END_RUNG
   RUNG wire#w1
      Contact( "Unit1.Em7.ControlNodes".jellyRollWinder."step".transition1[510] )
      { S7_Templates := "time_type := Time" } #statTonTime[510].TON(pt := T#300ms, et =>)
      Move(in := #JOB_5_STEP_11, out1 => "Unit1.Em7.ControlNodes".jellyRollWinder.sequence.status.nextStep)
   END_RUNG
   // the same network as SCL:
   #_w1 := ("Unit1.Em7.ControlNodes".jellyRollWinder.sequence.status.currentStep = #JOB_5_STEP_10) AND "Unit1.Em7.ControlNodes".jellyRollWinder.sequence.status.seqActive;
   "Unit1.Em7.ControlNodes".jellyRollWinder."step".action1[510] := #_w1 AND NOT #FALSE;
   "Unit1.Em7.ControlNodes".jellyRollWinder."step".transition1[510] := #_w1 AND "Unit1.Em7.ControlNodes".cm.softCam.jrWinderAxisB.angle450.inPos AND "Unit1.Em7.ControlNodes".cm.softCam.jrPusherAxisZ.verticalPos.inPos;
   #statTonTime[510].TON(IN := #_w1 AND "Unit1.Em7.ControlNodes".jellyRollWinder."step".transition1[510],
                         PT := T#300ms);
   IF #statTonTime[510].Q THEN
       "Unit1.Em7.ControlNodes".jellyRollWinder.sequence.status.nextStep := #JOB_5_STEP_11;
   END_IF;
END_REGION

REGION Network 36: Step[511] : Winder B-Axis 540 Angle Pos / Pusher Z-Axis Horizon Pos
   RUNG wire#powerrail
      { S7_Templates := "SrcType := DInt" } EQ_Contact(in1 := "Unit1.Em7.ControlNodes".jellyRollWinder.sequence.status.currentStep, in2 := #JOB_5_STEP_11)
      Contact( "Unit1.Em7.ControlNodes".jellyRollWinder.sequence.status.seqActive )
      wire#w1
      I_Contact( #FALSE )
      Coil( "Unit1.Em7.ControlNodes".jellyRollWinder."step".action1[511] )
   END_RUNG
   RUNG wire#w1
      Contact( "Unit1.Em7.ControlNodes".cm.softCam.jrWinderAxisB.angle540.inPos )
      Contact( "Unit1.Em7.ControlNodes".cm.softCam.jrPusherAxisZ.horizonPos.inPos )
      Coil( "Unit1.Em7.ControlNodes".jellyRollWinder."step".transition1[511] )
   END_RUNG
   RUNG wire#w1
      Contact( "Unit1.Em7.ControlNodes".jellyRollWinder."step".transition1[511] )
      { S7_Templates := "time_type := Time" } #statTonTime[511].TON(pt := T#300ms, et =>)
      Move(in := #JOB_5_STEP_90, out1 => "Unit1.Em7.ControlNodes".jellyRollWinder.sequence.status.nextStep)
   END_RUNG
   // the same network as SCL:
   #_w1 := ("Unit1.Em7.ControlNodes".jellyRollWinder.sequence.status.currentStep = #JOB_5_STEP_11) AND "Unit1.Em7.ControlNodes".jellyRollWinder.sequence.status.seqActive;
   "Unit1.Em7.ControlNodes".jellyRollWinder."step".action1[511] := #_w1 AND NOT #FALSE;
   "Unit1.Em7.ControlNodes".jellyRollWinder."step".transition1[511] := #_w1 AND "Unit1.Em7.ControlNodes".cm.softCam.jrWinderAxisB.angle540.inPos AND "Unit1.Em7.ControlNodes".cm.softCam.jrPusherAxisZ.horizonPos.inPos;
   #statTonTime[511].TON(IN := #_w1 AND "Unit1.Em7.ControlNodes".jellyRollWinder."step".transition1[511],
                         PT := T#300ms);
   IF #statTonTime[511].Q THEN
       "Unit1.Em7.ControlNodes".jellyRollWinder.sequence.status.nextStep := #JOB_5_STEP_90;
   END_IF;
END_REGION

REGION Network 37: Step[590] : Job[5] Step End
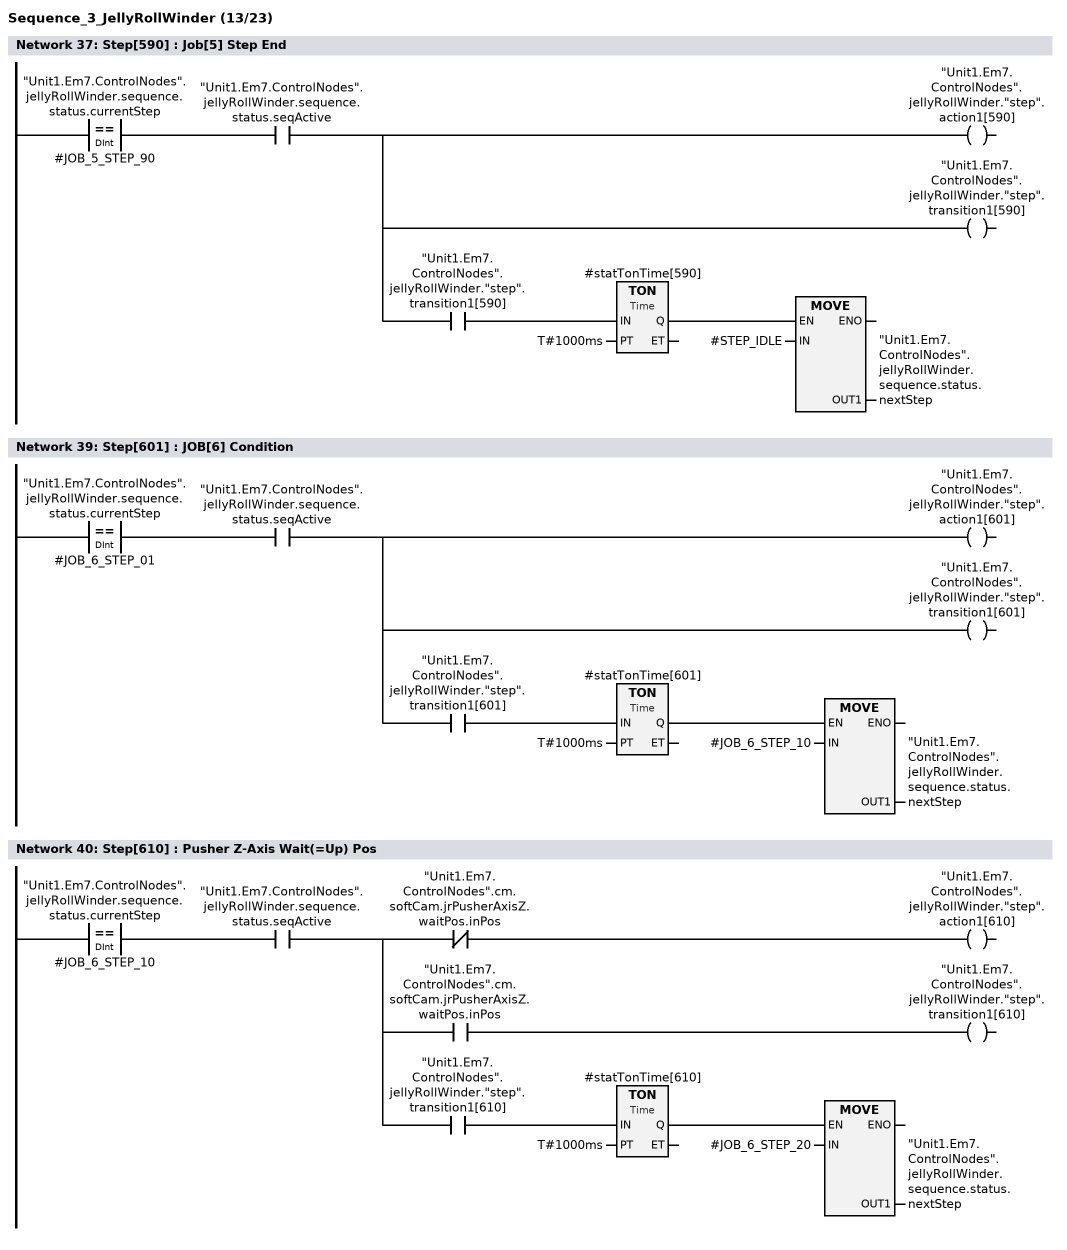
   RUNG wire#powerrail
      { S7_Templates := "SrcType := DInt" } EQ_Contact(in1 := "Unit1.Em7.ControlNodes".jellyRollWinder.sequence.status.currentStep, in2 := #JOB_5_STEP_90)
      Contact( "Unit1.Em7.ControlNodes".jellyRollWinder.sequence.status.seqActive )
      wire#w1
      Coil( "Unit1.Em7.ControlNodes".jellyRollWinder."step".action1[590] )
   END_RUNG
   RUNG wire#w1
      Coil( "Unit1.Em7.ControlNodes".jellyRollWinder."step".transition1[590] )
   END_RUNG
   RUNG wire#w1
      Contact( "Unit1.Em7.ControlNodes".jellyRollWinder."step".transition1[590] )
      { S7_Templates := "time_type := Time" } #statTonTime[590].TON(pt := T#1000ms, et =>)
      Move(in := #STEP_IDLE, out1 => "Unit1.Em7.ControlNodes".jellyRollWinder.sequence.status.nextStep)
   END_RUNG
   // the same network as SCL:
   "Unit1.Em7.ControlNodes".jellyRollWinder."step".action1[590] := ("Unit1.Em7.ControlNodes".jellyRollWinder.sequence.status.currentStep = #JOB_5_STEP_90) AND "Unit1.Em7.ControlNodes".jellyRollWinder.sequence.status.seqActive;
   "Unit1.Em7.ControlNodes".jellyRollWinder."step".transition1[590] := ("Unit1.Em7.ControlNodes".jellyRollWinder.sequence.status.currentStep = #JOB_5_STEP_90) AND "Unit1.Em7.ControlNodes".jellyRollWinder.sequence.status.seqActive;
   #statTonTime[590].TON(IN := ("Unit1.Em7.ControlNodes".jellyRollWinder.sequence.status.currentStep = #JOB_5_STEP_90) AND "Unit1.Em7.ControlNodes".jellyRollWinder.sequence.status.seqActive AND "Unit1.Em7.ControlNodes".jellyRollWinder."step".transition1[590],
                         PT := T#1000ms);
   IF #statTonTime[590].Q THEN
       "Unit1.Em7.ControlNodes".jellyRollWinder.sequence.status.nextStep := #STEP_IDLE;
   END_IF;
END_REGION

REGION Network 38: *************** JOB[6] Unload ************************
END_REGION

REGION Network 39: Step[601] : JOB[6] Condition
   RUNG wire#powerrail
      { S7_Templates := "SrcType := DInt" } EQ_Contact(in1 := "Unit1.Em7.ControlNodes".jellyRollWinder.sequence.status.currentStep, in2 := #JOB_6_STEP_01)
      Contact( "Unit1.Em7.ControlNodes".jellyRollWinder.sequence.status.seqActive )
      wire#w1
      Coil( "Unit1.Em7.ControlNodes".jellyRollWinder."step".action1[601] )
   END_RUNG
   RUNG wire#w1
      Coil( "Unit1.Em7.ControlNodes".jellyRollWinder."step".transition1[601] )
   END_RUNG
   RUNG wire#w1
      Contact( "Unit1.Em7.ControlNodes".jellyRollWinder."step".transition1[601] )
      { S7_Templates := "time_type := Time" } #statTonTime[601].TON(pt := T#1000ms, et =>)
      Move(in := #JOB_6_STEP_10, out1 => "Unit1.Em7.ControlNodes".jellyRollWinder.sequence.status.nextStep)
   END_RUNG
   // the same network as SCL:
   "Unit1.Em7.ControlNodes".jellyRollWinder."step".action1[601] := ("Unit1.Em7.ControlNodes".jellyRollWinder.sequence.status.currentStep = #JOB_6_STEP_01) AND "Unit1.Em7.ControlNodes".jellyRollWinder.sequence.status.seqActive;
   "Unit1.Em7.ControlNodes".jellyRollWinder."step".transition1[601] := ("Unit1.Em7.ControlNodes".jellyRollWinder.sequence.status.currentStep = #JOB_6_STEP_01) AND "Unit1.Em7.ControlNodes".jellyRollWinder.sequence.status.seqActive;
   #statTonTime[601].TON(IN := ("Unit1.Em7.ControlNodes".jellyRollWinder.sequence.status.currentStep = #JOB_6_STEP_01) AND "Unit1.Em7.ControlNodes".jellyRollWinder.sequence.status.seqActive AND "Unit1.Em7.ControlNodes".jellyRollWinder."step".transition1[601],
                         PT := T#1000ms);
   IF #statTonTime[601].Q THEN
       "Unit1.Em7.ControlNodes".jellyRollWinder.sequence.status.nextStep := #JOB_6_STEP_10;
   END_IF;
END_REGION

REGION Network 40: Step[610] : Pusher Z-Axis Wait(=Up) Pos
   RUNG wire#powerrail
      { S7_Templates := "SrcType := DInt" } EQ_Contact(in1 := "Unit1.Em7.ControlNodes".jellyRollWinder.sequence.status.currentStep, in2 := #JOB_6_STEP_10)
      Contact( "Unit1.Em7.ControlNodes".jellyRollWinder.sequence.status.seqActive )
      wire#w1
      I_Contact( "Unit1.Em7.ControlNodes".cm.softCam.jrPusherAxisZ.waitPos.inPos )
      Coil( "Unit1.Em7.ControlNodes".jellyRollWinder."step".action1[610] )
   END_RUNG
   RUNG wire#w1
      Contact( "Unit1.Em7.ControlNodes".cm.softCam.jrPusherAxisZ.waitPos.inPos )
      Coil( "Unit1.Em7.ControlNodes".jellyRollWinder."step".transition1[610] )
   END_RUNG
   RUNG wire#w1
      Contact( "Unit1.Em7.ControlNodes".jellyRollWinder."step".transition1[610] )
      { S7_Templates := "time_type := Time" } #statTonTime[610].TON(pt := T#1000ms, et =>)
      Move(in := #JOB_6_STEP_20, out1 => "Unit1.Em7.ControlNodes".jellyRollWinder.sequence.status.nextStep)
   END_RUNG
   // the same network as SCL:
   #_w1 := ("Unit1.Em7.ControlNodes".jellyRollWinder.sequence.status.currentStep = #JOB_6_STEP_10) AND "Unit1.Em7.ControlNodes".jellyRollWinder.sequence.status.seqActive;
   "Unit1.Em7.ControlNodes".jellyRollWinder."step".action1[610] := #_w1 AND NOT "Unit1.Em7.ControlNodes".cm.softCam.jrPusherAxisZ.waitPos.inPos;
   "Unit1.Em7.ControlNodes".jellyRollWinder."step".transition1[610] := #_w1 AND "Unit1.Em7.ControlNodes".cm.softCam.jrPusherAxisZ.waitPos.inPos;
   #statTonTime[610].TON(IN := #_w1 AND "Unit1.Em7.ControlNodes".jellyRollWinder."step".transition1[610],
                         PT := T#1000ms);
   IF #statTonTime[610].Q THEN
       "Unit1.Em7.ControlNodes".jellyRollWinder.sequence.status.nextStep := #JOB_6_STEP_20;
   END_IF;
END_REGION

REGION Network 41: Step[620] : Pusehr Backward
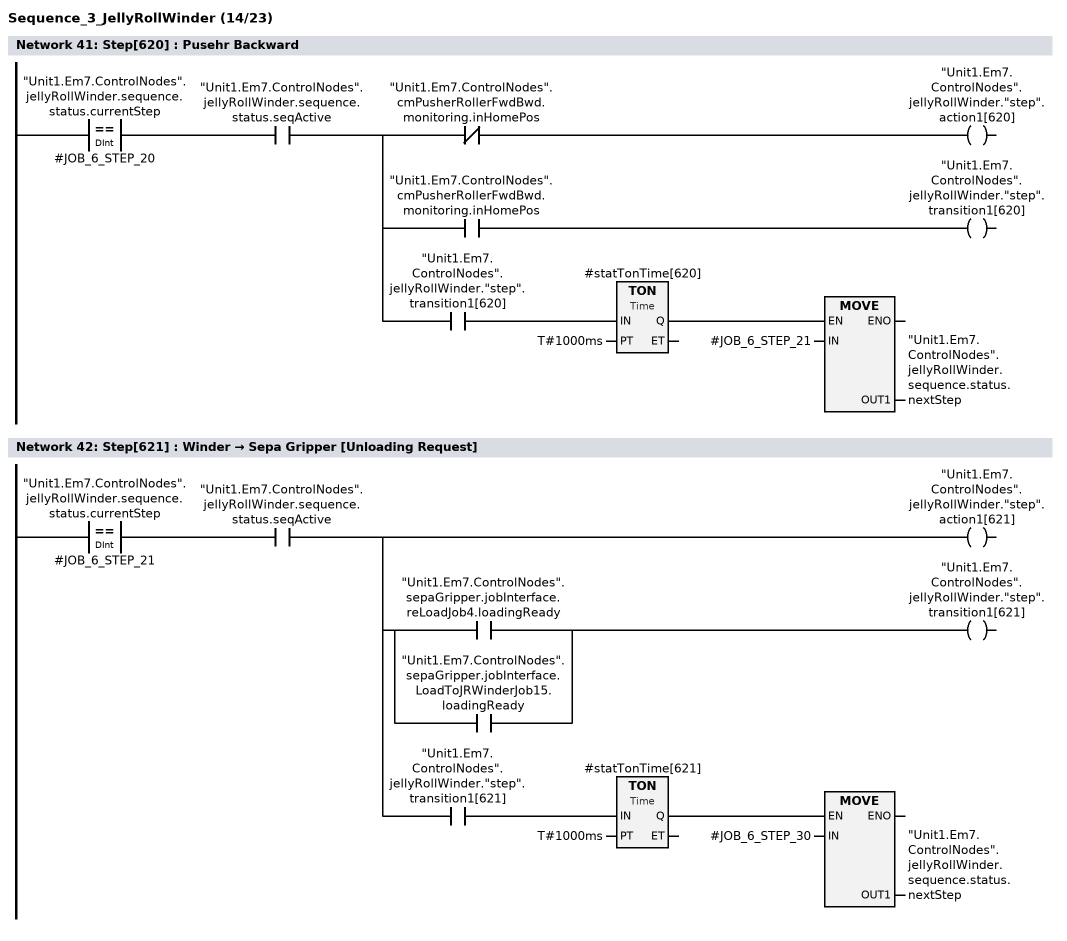
   RUNG wire#powerrail
      { S7_Templates := "SrcType := DInt" } EQ_Contact(in1 := "Unit1.Em7.ControlNodes".jellyRollWinder.sequence.status.currentStep, in2 := #JOB_6_STEP_20)
      Contact( "Unit1.Em7.ControlNodes".jellyRollWinder.sequence.status.seqActive )
      wire#w1
      I_Contact( "Unit1.Em7.ControlNodes".cmPusherRollerFwdBwd.monitoring.inHomePos )
      Coil( "Unit1.Em7.ControlNodes".jellyRollWinder."step".action1[620] )
   END_RUNG
   RUNG wire#w1
      Contact( "Unit1.Em7.ControlNodes".cmPusherRollerFwdBwd.monitoring.inHomePos )
      Coil( "Unit1.Em7.ControlNodes".jellyRollWinder."step".transition1[620] )
   END_RUNG
   RUNG wire#w1
      Contact( "Unit1.Em7.ControlNodes".jellyRollWinder."step".transition1[620] )
      { S7_Templates := "time_type := Time" } #statTonTime[620].TON(pt := T#1000ms, et =>)
      Move(in := #JOB_6_STEP_21, out1 => "Unit1.Em7.ControlNodes".jellyRollWinder.sequence.status.nextStep)
   END_RUNG
   // the same network as SCL:
   #_w1 := ("Unit1.Em7.ControlNodes".jellyRollWinder.sequence.status.currentStep = #JOB_6_STEP_20) AND "Unit1.Em7.ControlNodes".jellyRollWinder.sequence.status.seqActive;
   "Unit1.Em7.ControlNodes".jellyRollWinder."step".action1[620] := #_w1 AND NOT "Unit1.Em7.ControlNodes".cmPusherRollerFwdBwd.monitoring.inHomePos;
   "Unit1.Em7.ControlNodes".jellyRollWinder."step".transition1[620] := #_w1 AND "Unit1.Em7.ControlNodes".cmPusherRollerFwdBwd.monitoring.inHomePos;
   #statTonTime[620].TON(IN := #_w1 AND "Unit1.Em7.ControlNodes".jellyRollWinder."step".transition1[620],
                         PT := T#1000ms);
   IF #statTonTime[620].Q THEN
       "Unit1.Em7.ControlNodes".jellyRollWinder.sequence.status.nextStep := #JOB_6_STEP_21;
   END_IF;
END_REGION

REGION Network 42: Step[621] : Winder → Sepa Gripper [Unloading Request]
   RUNG wire#powerrail
      { S7_Templates := "SrcType := DInt" } EQ_Contact(in1 := "Unit1.Em7.ControlNodes".jellyRollWinder.sequence.status.currentStep, in2 := #JOB_6_STEP_21)
      Contact( "Unit1.Em7.ControlNodes".jellyRollWinder.sequence.status.seqActive )
      wire#w1
      Coil( "Unit1.Em7.ControlNodes".jellyRollWinder."step".action1[621] )
   END_RUNG
   RUNG wire#w1
      Contact( "Unit1.Em7.ControlNodes".sepaGripper.jobInterface.reLoadJob4.loadingReady )
      wire#w2
      Coil( "Unit1.Em7.ControlNodes".jellyRollWinder."step".transition1[621] )
   END_RUNG
   RUNG wire#w1
      Contact( "Unit1.Em7.ControlNodes".sepaGripper.jobInterface.LoadToJRWinderJob15.loadingReady )
   END_RUNG wire#w2
   RUNG wire#w1
      Contact( "Unit1.Em7.ControlNodes".jellyRollWinder."step".transition1[621] )
      { S7_Templates := "time_type := Time" } #statTonTime[621].TON(pt := T#1000ms, et =>)
      Move(in := #JOB_6_STEP_30, out1 => "Unit1.Em7.ControlNodes".jellyRollWinder.sequence.status.nextStep)
   END_RUNG
   // the same network as SCL:
   "Unit1.Em7.ControlNodes".jellyRollWinder."step".action1[621] := ("Unit1.Em7.ControlNodes".jellyRollWinder.sequence.status.currentStep = #JOB_6_STEP_21) AND "Unit1.Em7.ControlNodes".jellyRollWinder.sequence.status.seqActive;
   "Unit1.Em7.ControlNodes".jellyRollWinder."step".transition1[621] := ("Unit1.Em7.ControlNodes".jellyRollWinder.sequence.status.currentStep = #JOB_6_STEP_21) AND "Unit1.Em7.ControlNodes".jellyRollWinder.sequence.status.seqActive AND ("Unit1.Em7.ControlNodes".sepaGripper.jobInterface.reLoadJob4.loadingReady OR "Unit1.Em7.ControlNodes".sepaGripper.jobInterface.LoadToJRWinderJob15.loadingReady);
   #statTonTime[621].TON(IN := ("Unit1.Em7.ControlNodes".jellyRollWinder.sequence.status.currentStep = #JOB_6_STEP_21) AND "Unit1.Em7.ControlNodes".jellyRollWinder.sequence.status.seqActive AND "Unit1.Em7.ControlNodes".jellyRollWinder."step".transition1[621],
                         PT := T#1000ms);
   IF #statTonTime[621].Q THEN
       "Unit1.Em7.ControlNodes".jellyRollWinder.sequence.status.nextStep := #JOB_6_STEP_30;
   END_IF;
END_REGION

REGION Network 43: Step[630] : Winder Open
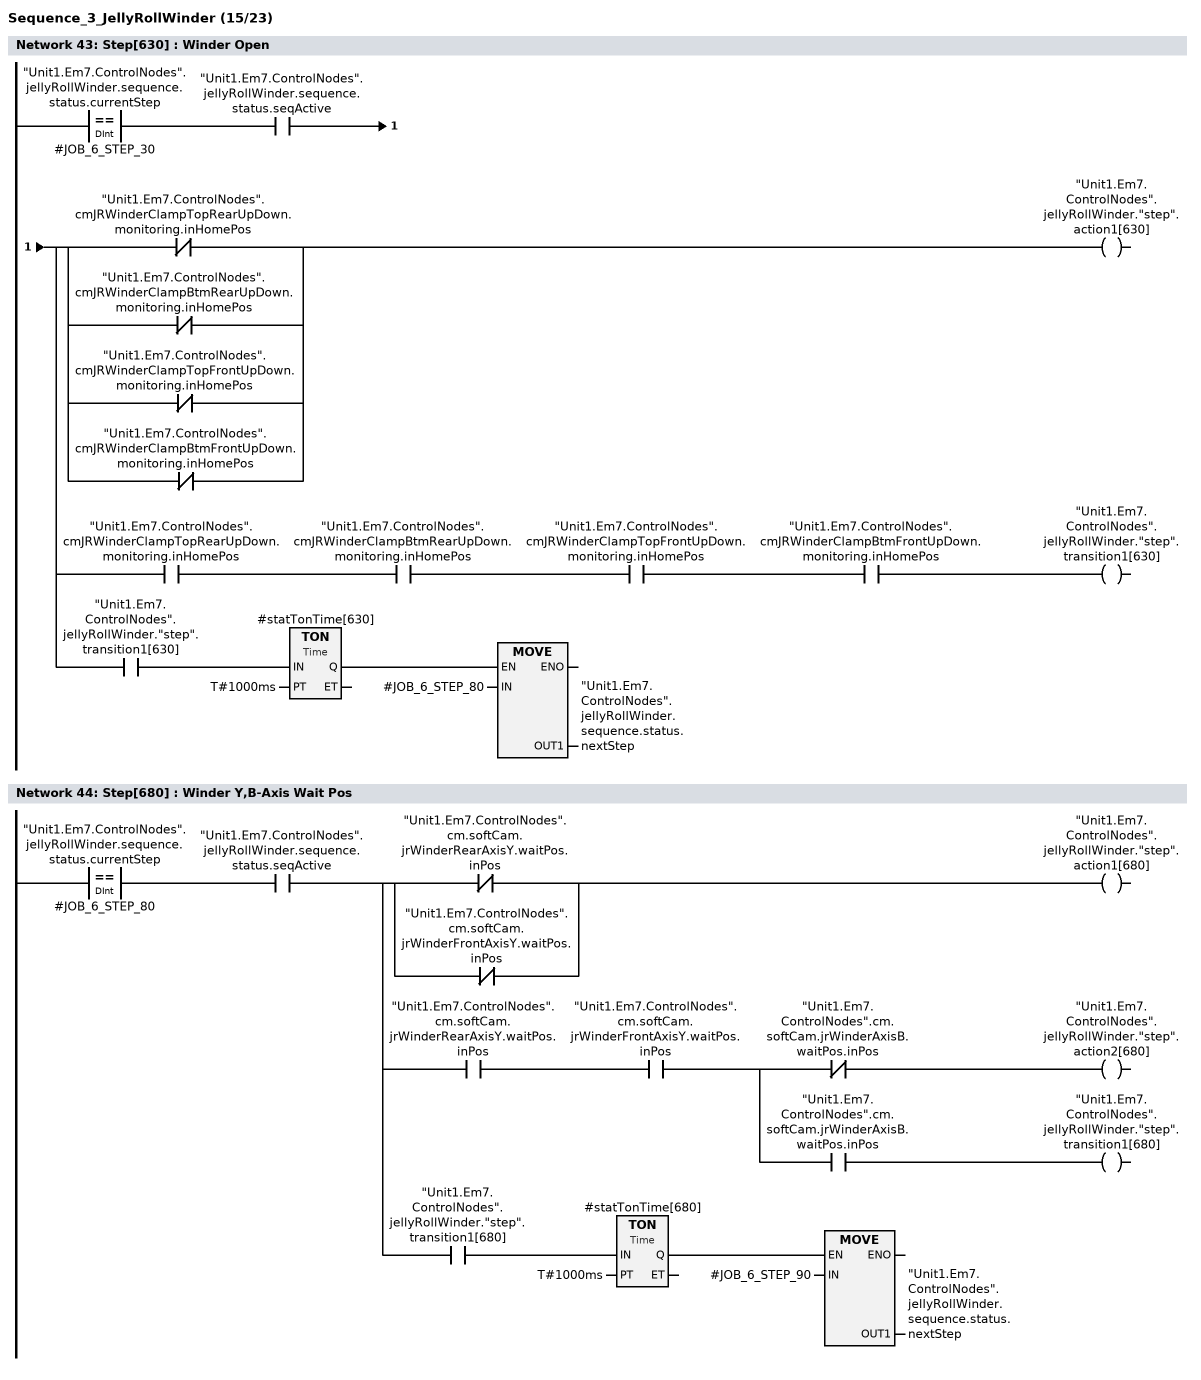
   RUNG wire#powerrail
      { S7_Templates := "SrcType := DInt" } EQ_Contact(in1 := "Unit1.Em7.ControlNodes".jellyRollWinder.sequence.status.currentStep, in2 := #JOB_6_STEP_30)
      Contact( "Unit1.Em7.ControlNodes".jellyRollWinder.sequence.status.seqActive )
      wire#w1
      I_Contact( "Unit1.Em7.ControlNodes".cmJRWinderClampTopRearUpDown.monitoring.inHomePos )
      wire#w2
      Coil( "Unit1.Em7.ControlNodes".jellyRollWinder."step".action1[630] )
   END_RUNG
   RUNG wire#w1
      I_Contact( "Unit1.Em7.ControlNodes".cmJRWinderClampBtmRearUpDown.monitoring.inHomePos )
   END_RUNG wire#w2
   RUNG wire#w1
      I_Contact( "Unit1.Em7.ControlNodes".cmJRWinderClampTopFrontUpDown.monitoring.inHomePos )
   END_RUNG wire#w2
   RUNG wire#w1
      I_Contact( "Unit1.Em7.ControlNodes".cmJRWinderClampBtmFrontUpDown.monitoring.inHomePos )
   END_RUNG wire#w2
   RUNG wire#w1
      Contact( "Unit1.Em7.ControlNodes".cmJRWinderClampTopRearUpDown.monitoring.inHomePos )
      Contact( "Unit1.Em7.ControlNodes".cmJRWinderClampBtmRearUpDown.monitoring.inHomePos )
      Contact( "Unit1.Em7.ControlNodes".cmJRWinderClampTopFrontUpDown.monitoring.inHomePos )
      Contact( "Unit1.Em7.ControlNodes".cmJRWinderClampBtmFrontUpDown.monitoring.inHomePos )
      Coil( "Unit1.Em7.ControlNodes".jellyRollWinder."step".transition1[630] )
   END_RUNG
   RUNG wire#w1
      Contact( "Unit1.Em7.ControlNodes".jellyRollWinder."step".transition1[630] )
      { S7_Templates := "time_type := Time" } #statTonTime[630].TON(pt := T#1000ms, et =>)
      Move(in := #JOB_6_STEP_80, out1 => "Unit1.Em7.ControlNodes".jellyRollWinder.sequence.status.nextStep)
   END_RUNG
   // the same network as SCL:
   #_w1 := ("Unit1.Em7.ControlNodes".jellyRollWinder.sequence.status.currentStep = #JOB_6_STEP_30) AND "Unit1.Em7.ControlNodes".jellyRollWinder.sequence.status.seqActive;
   "Unit1.Em7.ControlNodes".jellyRollWinder."step".action1[630] := #_w1 AND (NOT "Unit1.Em7.ControlNodes".cmJRWinderClampTopRearUpDown.monitoring.inHomePos OR NOT "Unit1.Em7.ControlNodes".cmJRWinderClampBtmRearUpDown.monitoring.inHomePos OR NOT "Unit1.Em7.ControlNodes".cmJRWinderClampTopFrontUpDown.monitoring.inHomePos OR NOT "Unit1.Em7.ControlNodes".cmJRWinderClampBtmFrontUpDown.monitoring.inHomePos);
   "Unit1.Em7.ControlNodes".jellyRollWinder."step".transition1[630] := #_w1 AND "Unit1.Em7.ControlNodes".cmJRWinderClampTopRearUpDown.monitoring.inHomePos AND "Unit1.Em7.ControlNodes".cmJRWinderClampBtmRearUpDown.monitoring.inHomePos AND "Unit1.Em7.ControlNodes".cmJRWinderClampTopFrontUpDown.monitoring.inHomePos AND "Unit1.Em7.ControlNodes".cmJRWinderClampBtmFrontUpDown.monitoring.inHomePos;
   #statTonTime[630].TON(IN := #_w1 AND "Unit1.Em7.ControlNodes".jellyRollWinder."step".transition1[630],
                         PT := T#1000ms);
   IF #statTonTime[630].Q THEN
       "Unit1.Em7.ControlNodes".jellyRollWinder.sequence.status.nextStep := #JOB_6_STEP_80;
   END_IF;
END_REGION

REGION Network 44: Step[680] : Winder Y,B-Axis Wait Pos
   RUNG wire#powerrail
      { S7_Templates := "SrcType := DInt" } EQ_Contact(in1 := "Unit1.Em7.ControlNodes".jellyRollWinder.sequence.status.currentStep, in2 := #JOB_6_STEP_80)
      Contact( "Unit1.Em7.ControlNodes".jellyRollWinder.sequence.status.seqActive )
      wire#w1
      I_Contact( "Unit1.Em7.ControlNodes".cm.softCam.jrWinderRearAxisY.waitPos.inPos )
      wire#w2
      Coil( "Unit1.Em7.ControlNodes".jellyRollWinder."step".action1[680] )
   END_RUNG
   RUNG wire#w1
      I_Contact( "Unit1.Em7.ControlNodes".cm.softCam.jrWinderFrontAxisY.waitPos.inPos )
   END_RUNG wire#w2
   RUNG wire#w1
      Contact( "Unit1.Em7.ControlNodes".cm.softCam.jrWinderRearAxisY.waitPos.inPos )
      Contact( "Unit1.Em7.ControlNodes".cm.softCam.jrWinderFrontAxisY.waitPos.inPos )
      wire#w3
      I_Contact( "Unit1.Em7.ControlNodes".cm.softCam.jrWinderAxisB.waitPos.inPos )
      Coil( "Unit1.Em7.ControlNodes".jellyRollWinder."step".action2[680] )
   END_RUNG
   RUNG wire#w3
      Contact( "Unit1.Em7.ControlNodes".cm.softCam.jrWinderAxisB.waitPos.inPos )
      Coil( "Unit1.Em7.ControlNodes".jellyRollWinder."step".transition1[680] )
   END_RUNG
   RUNG wire#w1
      Contact( "Unit1.Em7.ControlNodes".jellyRollWinder."step".transition1[680] )
      { S7_Templates := "time_type := Time" } #statTonTime[680].TON(pt := T#1000ms, et =>)
      Move(in := #JOB_6_STEP_90, out1 => "Unit1.Em7.ControlNodes".jellyRollWinder.sequence.status.nextStep)
   END_RUNG
   // the same network as SCL:
   #_w1 := ("Unit1.Em7.ControlNodes".jellyRollWinder.sequence.status.currentStep = #JOB_6_STEP_80) AND "Unit1.Em7.ControlNodes".jellyRollWinder.sequence.status.seqActive;
   "Unit1.Em7.ControlNodes".jellyRollWinder."step".action1[680] := #_w1 AND (NOT "Unit1.Em7.ControlNodes".cm.softCam.jrWinderRearAxisY.waitPos.inPos OR NOT "Unit1.Em7.ControlNodes".cm.softCam.jrWinderFrontAxisY.waitPos.inPos);
   #_w2 := #_w1 AND "Unit1.Em7.ControlNodes".cm.softCam.jrWinderRearAxisY.waitPos.inPos AND "Unit1.Em7.ControlNodes".cm.softCam.jrWinderFrontAxisY.waitPos.inPos;
   "Unit1.Em7.ControlNodes".jellyRollWinder."step".action2[680] := #_w2 AND NOT "Unit1.Em7.ControlNodes".cm.softCam.jrWinderAxisB.waitPos.inPos;
   "Unit1.Em7.ControlNodes".jellyRollWinder."step".transition1[680] := #_w2 AND "Unit1.Em7.ControlNodes".cm.softCam.jrWinderAxisB.waitPos.inPos;
   #statTonTime[680].TON(IN := #_w1 AND "Unit1.Em7.ControlNodes".jellyRollWinder."step".transition1[680],
                         PT := T#1000ms);
   IF #statTonTime[680].Q THEN
       "Unit1.Em7.ControlNodes".jellyRollWinder.sequence.status.nextStep := #JOB_6_STEP_90;
   END_IF;
END_REGION

REGION Network 45: Step[690] : Job[6] Step End
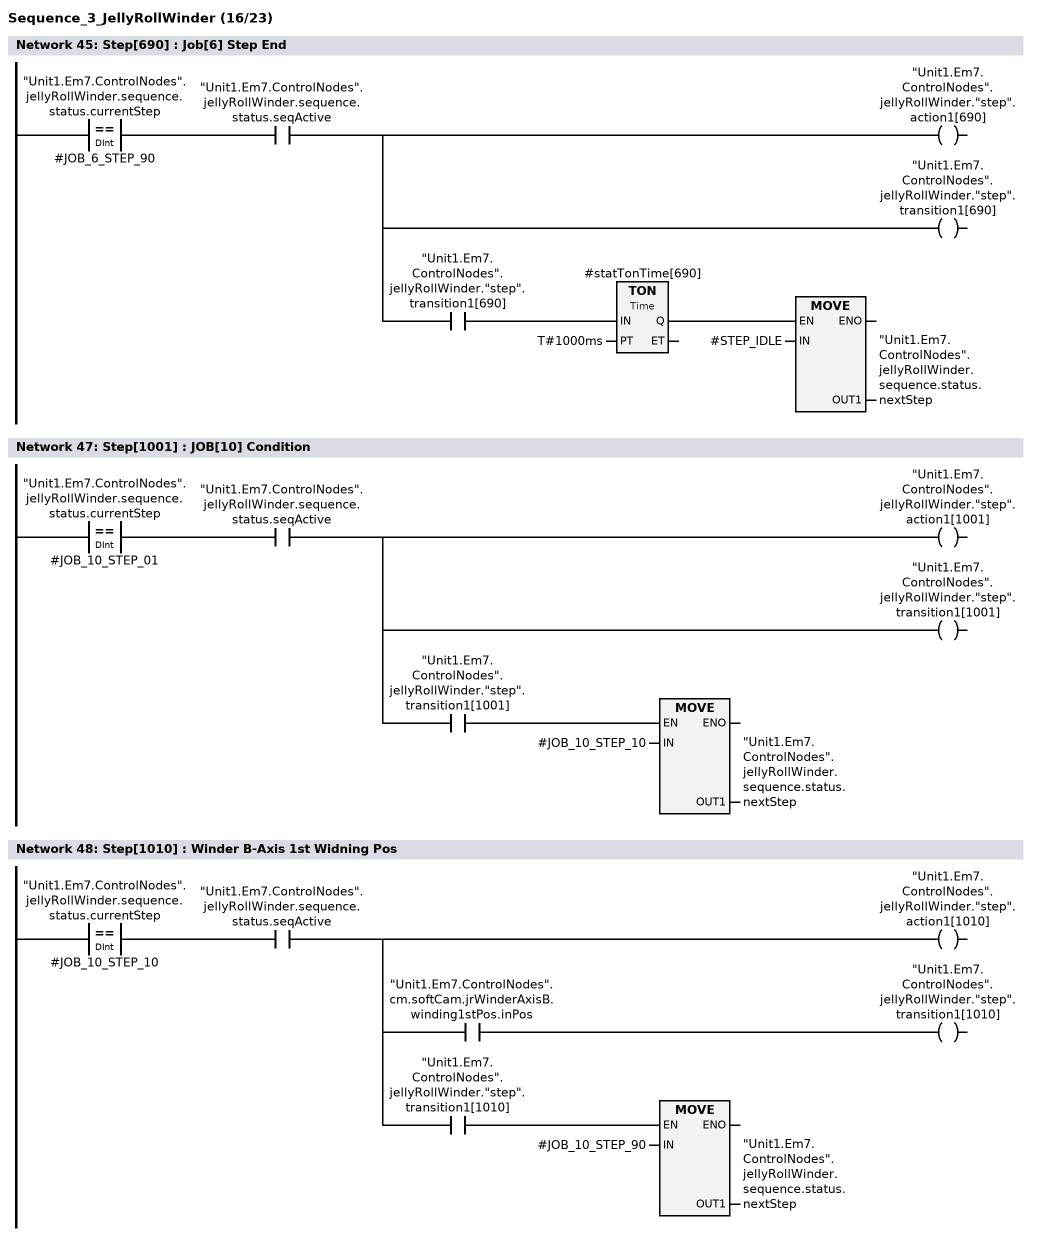
   RUNG wire#powerrail
      { S7_Templates := "SrcType := DInt" } EQ_Contact(in1 := "Unit1.Em7.ControlNodes".jellyRollWinder.sequence.status.currentStep, in2 := #JOB_6_STEP_90)
      Contact( "Unit1.Em7.ControlNodes".jellyRollWinder.sequence.status.seqActive )
      wire#w1
      Coil( "Unit1.Em7.ControlNodes".jellyRollWinder."step".action1[690] )
   END_RUNG
   RUNG wire#w1
      Coil( "Unit1.Em7.ControlNodes".jellyRollWinder."step".transition1[690] )
   END_RUNG
   RUNG wire#w1
      Contact( "Unit1.Em7.ControlNodes".jellyRollWinder."step".transition1[690] )
      { S7_Templates := "time_type := Time" } #statTonTime[690].TON(pt := T#1000ms, et =>)
      Move(in := #STEP_IDLE, out1 => "Unit1.Em7.ControlNodes".jellyRollWinder.sequence.status.nextStep)
   END_RUNG
   // the same network as SCL:
   "Unit1.Em7.ControlNodes".jellyRollWinder."step".action1[690] := ("Unit1.Em7.ControlNodes".jellyRollWinder.sequence.status.currentStep = #JOB_6_STEP_90) AND "Unit1.Em7.ControlNodes".jellyRollWinder.sequence.status.seqActive;
   "Unit1.Em7.ControlNodes".jellyRollWinder."step".transition1[690] := ("Unit1.Em7.ControlNodes".jellyRollWinder.sequence.status.currentStep = #JOB_6_STEP_90) AND "Unit1.Em7.ControlNodes".jellyRollWinder.sequence.status.seqActive;
   #statTonTime[690].TON(IN := ("Unit1.Em7.ControlNodes".jellyRollWinder.sequence.status.currentStep = #JOB_6_STEP_90) AND "Unit1.Em7.ControlNodes".jellyRollWinder.sequence.status.seqActive AND "Unit1.Em7.ControlNodes".jellyRollWinder."step".transition1[690],
                         PT := T#1000ms);
   IF #statTonTime[690].Q THEN
       "Unit1.Em7.ControlNodes".jellyRollWinder.sequence.status.nextStep := #STEP_IDLE;
   END_IF;
END_REGION

REGION Network 46: *************** JOB[10] Cam 1st Winding ************************
END_REGION

REGION Network 47: Step[1001] : JOB[10] Condition
   RUNG wire#powerrail
      { S7_Templates := "SrcType := DInt" } EQ_Contact(in1 := "Unit1.Em7.ControlNodes".jellyRollWinder.sequence.status.currentStep, in2 := #JOB_10_STEP_01)
      Contact( "Unit1.Em7.ControlNodes".jellyRollWinder.sequence.status.seqActive )
      wire#w1
      Coil( "Unit1.Em7.ControlNodes".jellyRollWinder."step".action1[1001] )
   END_RUNG
   RUNG wire#w1
      Coil( "Unit1.Em7.ControlNodes".jellyRollWinder."step".transition1[1001] )
   END_RUNG
   RUNG wire#w1
      Contact( "Unit1.Em7.ControlNodes".jellyRollWinder."step".transition1[1001] )
      Move(in := #JOB_10_STEP_10, out1 => "Unit1.Em7.ControlNodes".jellyRollWinder.sequence.status.nextStep)
   END_RUNG
   // the same network as SCL:
   "Unit1.Em7.ControlNodes".jellyRollWinder."step".action1[1001] := ("Unit1.Em7.ControlNodes".jellyRollWinder.sequence.status.currentStep = #JOB_10_STEP_01) AND "Unit1.Em7.ControlNodes".jellyRollWinder.sequence.status.seqActive;
   "Unit1.Em7.ControlNodes".jellyRollWinder."step".transition1[1001] := ("Unit1.Em7.ControlNodes".jellyRollWinder.sequence.status.currentStep = #JOB_10_STEP_01) AND "Unit1.Em7.ControlNodes".jellyRollWinder.sequence.status.seqActive;
   IF ("Unit1.Em7.ControlNodes".jellyRollWinder.sequence.status.currentStep = #JOB_10_STEP_01) AND "Unit1.Em7.ControlNodes".jellyRollWinder.sequence.status.seqActive AND "Unit1.Em7.ControlNodes".jellyRollWinder."step".transition1[1001] THEN
       "Unit1.Em7.ControlNodes".jellyRollWinder.sequence.status.nextStep := #JOB_10_STEP_10;
   END_IF;
END_REGION

REGION Network 48: Step[1010] : Winder B-Axis 1st Widning Pos
   RUNG wire#powerrail
      { S7_Templates := "SrcType := DInt" } EQ_Contact(in1 := "Unit1.Em7.ControlNodes".jellyRollWinder.sequence.status.currentStep, in2 := #JOB_10_STEP_10)
      Contact( "Unit1.Em7.ControlNodes".jellyRollWinder.sequence.status.seqActive )
      wire#w1
      Coil( "Unit1.Em7.ControlNodes".jellyRollWinder."step".action1[1010] )
   END_RUNG
   RUNG wire#w1
      Contact( "Unit1.Em7.ControlNodes".cm.softCam.jrWinderAxisB.winding1stPos.inPos )
      Coil( "Unit1.Em7.ControlNodes".jellyRollWinder."step".transition1[1010] )
   END_RUNG
   RUNG wire#w1
      Contact( "Unit1.Em7.ControlNodes".jellyRollWinder."step".transition1[1010] )
      Move(in := #JOB_10_STEP_90, out1 => "Unit1.Em7.ControlNodes".jellyRollWinder.sequence.status.nextStep)
   END_RUNG
   // the same network as SCL:
   "Unit1.Em7.ControlNodes".jellyRollWinder."step".action1[1010] := ("Unit1.Em7.ControlNodes".jellyRollWinder.sequence.status.currentStep = #JOB_10_STEP_10) AND "Unit1.Em7.ControlNodes".jellyRollWinder.sequence.status.seqActive;
   "Unit1.Em7.ControlNodes".jellyRollWinder."step".transition1[1010] := ("Unit1.Em7.ControlNodes".jellyRollWinder.sequence.status.currentStep = #JOB_10_STEP_10) AND "Unit1.Em7.ControlNodes".jellyRollWinder.sequence.status.seqActive AND "Unit1.Em7.ControlNodes".cm.softCam.jrWinderAxisB.winding1stPos.inPos;
   IF ("Unit1.Em7.ControlNodes".jellyRollWinder.sequence.status.currentStep = #JOB_10_STEP_10) AND "Unit1.Em7.ControlNodes".jellyRollWinder.sequence.status.seqActive AND "Unit1.Em7.ControlNodes".jellyRollWinder."step".transition1[1010] THEN
       "Unit1.Em7.ControlNodes".jellyRollWinder.sequence.status.nextStep := #JOB_10_STEP_90;
   END_IF;
END_REGION

REGION Network 49: Step[1090] : Job[10] Step End
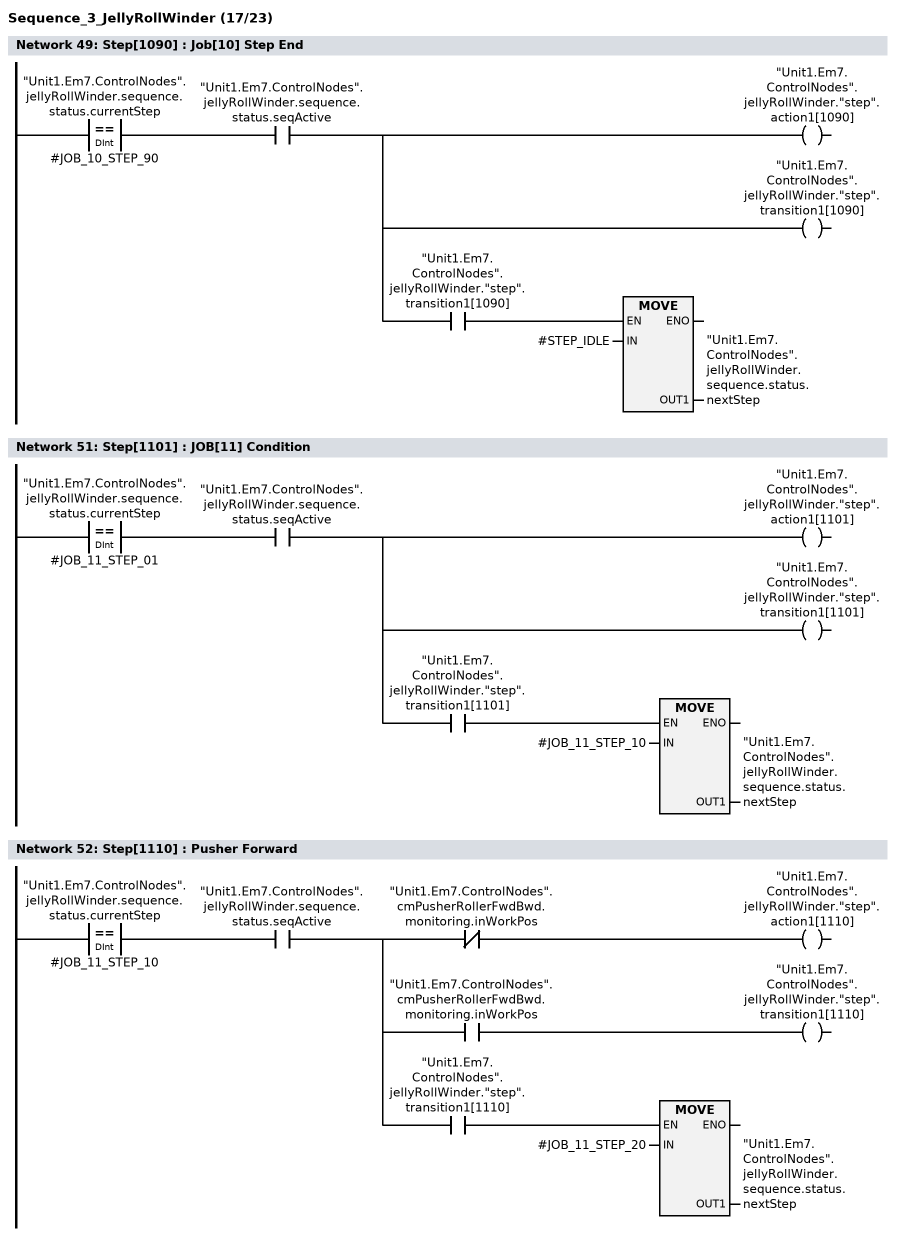
   RUNG wire#powerrail
      { S7_Templates := "SrcType := DInt" } EQ_Contact(in1 := "Unit1.Em7.ControlNodes".jellyRollWinder.sequence.status.currentStep, in2 := #JOB_10_STEP_90)
      Contact( "Unit1.Em7.ControlNodes".jellyRollWinder.sequence.status.seqActive )
      wire#w1
      Coil( "Unit1.Em7.ControlNodes".jellyRollWinder."step".action1[1090] )
   END_RUNG
   RUNG wire#w1
      Coil( "Unit1.Em7.ControlNodes".jellyRollWinder."step".transition1[1090] )
   END_RUNG
   RUNG wire#w1
      Contact( "Unit1.Em7.ControlNodes".jellyRollWinder."step".transition1[1090] )
      Move(in := #STEP_IDLE, out1 => "Unit1.Em7.ControlNodes".jellyRollWinder.sequence.status.nextStep)
   END_RUNG
   // the same network as SCL:
   "Unit1.Em7.ControlNodes".jellyRollWinder."step".action1[1090] := ("Unit1.Em7.ControlNodes".jellyRollWinder.sequence.status.currentStep = #JOB_10_STEP_90) AND "Unit1.Em7.ControlNodes".jellyRollWinder.sequence.status.seqActive;
   "Unit1.Em7.ControlNodes".jellyRollWinder."step".transition1[1090] := ("Unit1.Em7.ControlNodes".jellyRollWinder.sequence.status.currentStep = #JOB_10_STEP_90) AND "Unit1.Em7.ControlNodes".jellyRollWinder.sequence.status.seqActive;
   IF ("Unit1.Em7.ControlNodes".jellyRollWinder.sequence.status.currentStep = #JOB_10_STEP_90) AND "Unit1.Em7.ControlNodes".jellyRollWinder.sequence.status.seqActive AND "Unit1.Em7.ControlNodes".jellyRollWinder."step".transition1[1090] THEN
       "Unit1.Em7.ControlNodes".jellyRollWinder.sequence.status.nextStep := #STEP_IDLE;
   END_IF;
END_REGION

REGION Network 50: *************** JOB[11] Cam Pusher Ready ************************
END_REGION

REGION Network 51: Step[1101] : JOB[11] Condition
   RUNG wire#powerrail
      { S7_Templates := "SrcType := DInt" } EQ_Contact(in1 := "Unit1.Em7.ControlNodes".jellyRollWinder.sequence.status.currentStep, in2 := #JOB_11_STEP_01)
      Contact( "Unit1.Em7.ControlNodes".jellyRollWinder.sequence.status.seqActive )
      wire#w1
      Coil( "Unit1.Em7.ControlNodes".jellyRollWinder."step".action1[1101] )
   END_RUNG
   RUNG wire#w1
      Coil( "Unit1.Em7.ControlNodes".jellyRollWinder."step".transition1[1101] )
   END_RUNG
   RUNG wire#w1
      Contact( "Unit1.Em7.ControlNodes".jellyRollWinder."step".transition1[1101] )
      Move(in := #JOB_11_STEP_10, out1 => "Unit1.Em7.ControlNodes".jellyRollWinder.sequence.status.nextStep)
   END_RUNG
   // the same network as SCL:
   "Unit1.Em7.ControlNodes".jellyRollWinder."step".action1[1101] := ("Unit1.Em7.ControlNodes".jellyRollWinder.sequence.status.currentStep = #JOB_11_STEP_01) AND "Unit1.Em7.ControlNodes".jellyRollWinder.sequence.status.seqActive;
   "Unit1.Em7.ControlNodes".jellyRollWinder."step".transition1[1101] := ("Unit1.Em7.ControlNodes".jellyRollWinder.sequence.status.currentStep = #JOB_11_STEP_01) AND "Unit1.Em7.ControlNodes".jellyRollWinder.sequence.status.seqActive;
   IF ("Unit1.Em7.ControlNodes".jellyRollWinder.sequence.status.currentStep = #JOB_11_STEP_01) AND "Unit1.Em7.ControlNodes".jellyRollWinder.sequence.status.seqActive AND "Unit1.Em7.ControlNodes".jellyRollWinder."step".transition1[1101] THEN
       "Unit1.Em7.ControlNodes".jellyRollWinder.sequence.status.nextStep := #JOB_11_STEP_10;
   END_IF;
END_REGION

REGION Network 52: Step[1110] : Pusher Forward
   RUNG wire#powerrail
      { S7_Templates := "SrcType := DInt" } EQ_Contact(in1 := "Unit1.Em7.ControlNodes".jellyRollWinder.sequence.status.currentStep, in2 := #JOB_11_STEP_10)
      Contact( "Unit1.Em7.ControlNodes".jellyRollWinder.sequence.status.seqActive )
      wire#w1
      I_Contact( "Unit1.Em7.ControlNodes".cmPusherRollerFwdBwd.monitoring.inWorkPos )
      Coil( "Unit1.Em7.ControlNodes".jellyRollWinder."step".action1[1110] )
   END_RUNG
   RUNG wire#w1
      Contact( "Unit1.Em7.ControlNodes".cmPusherRollerFwdBwd.monitoring.inWorkPos )
      Coil( "Unit1.Em7.ControlNodes".jellyRollWinder."step".transition1[1110] )
   END_RUNG
   RUNG wire#w1
      Contact( "Unit1.Em7.ControlNodes".jellyRollWinder."step".transition1[1110] )
      Move(in := #JOB_11_STEP_20, out1 => "Unit1.Em7.ControlNodes".jellyRollWinder.sequence.status.nextStep)
   END_RUNG
   // the same network as SCL:
   #_w1 := ("Unit1.Em7.ControlNodes".jellyRollWinder.sequence.status.currentStep = #JOB_11_STEP_10) AND "Unit1.Em7.ControlNodes".jellyRollWinder.sequence.status.seqActive;
   "Unit1.Em7.ControlNodes".jellyRollWinder."step".action1[1110] := #_w1 AND NOT "Unit1.Em7.ControlNodes".cmPusherRollerFwdBwd.monitoring.inWorkPos;
   "Unit1.Em7.ControlNodes".jellyRollWinder."step".transition1[1110] := #_w1 AND "Unit1.Em7.ControlNodes".cmPusherRollerFwdBwd.monitoring.inWorkPos;
   IF #_w1 AND "Unit1.Em7.ControlNodes".jellyRollWinder."step".transition1[1110] THEN
       "Unit1.Em7.ControlNodes".jellyRollWinder.sequence.status.nextStep := #JOB_11_STEP_20;
   END_IF;
END_REGION

REGION Network 53: Step[1120] : Pusher Z-Axis Work(=Down) Pos
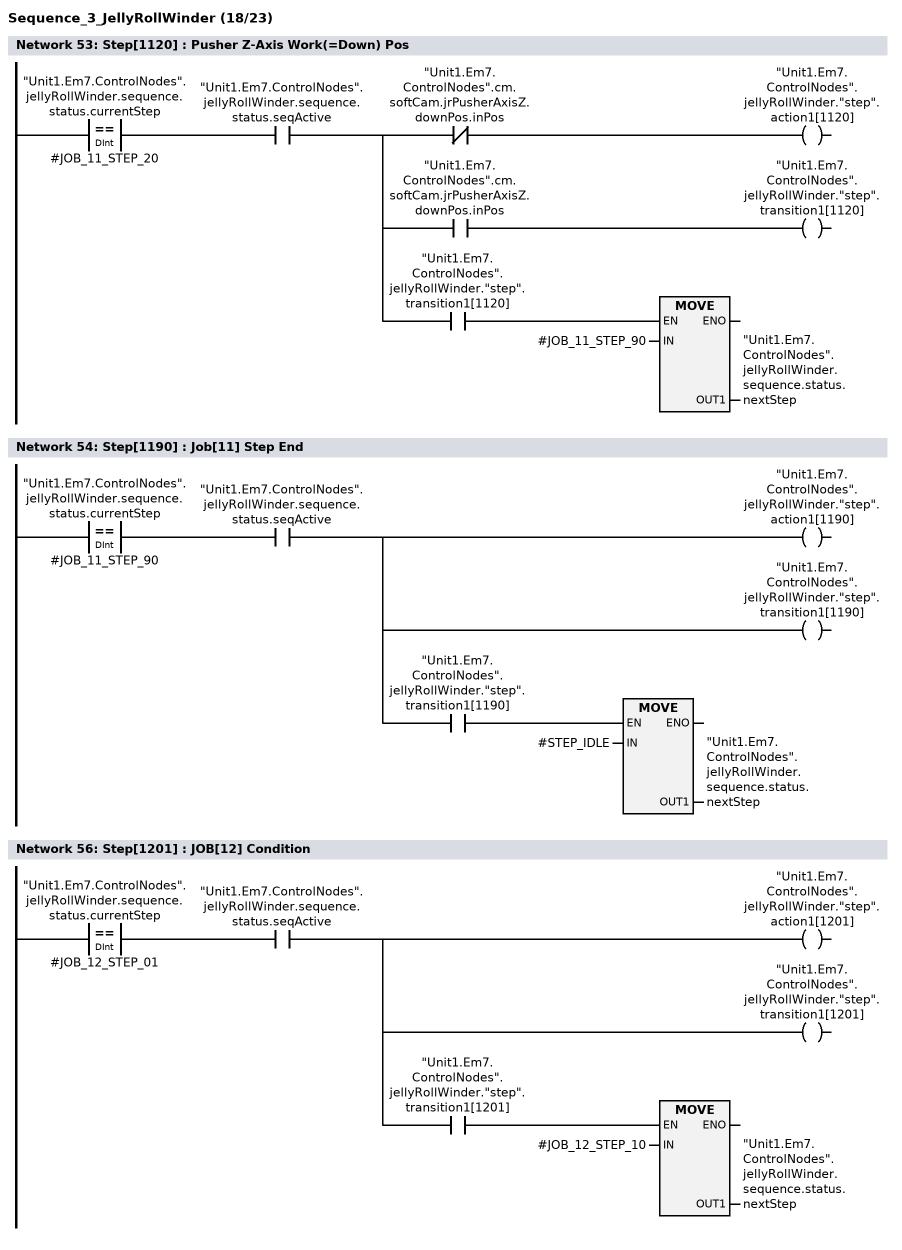
   RUNG wire#powerrail
      { S7_Templates := "SrcType := DInt" } EQ_Contact(in1 := "Unit1.Em7.ControlNodes".jellyRollWinder.sequence.status.currentStep, in2 := #JOB_11_STEP_20)
      Contact( "Unit1.Em7.ControlNodes".jellyRollWinder.sequence.status.seqActive )
      wire#w1
      I_Contact( "Unit1.Em7.ControlNodes".cm.softCam.jrPusherAxisZ.downPos.inPos )
      Coil( "Unit1.Em7.ControlNodes".jellyRollWinder."step".action1[1120] )
   END_RUNG
   RUNG wire#w1
      Contact( "Unit1.Em7.ControlNodes".cm.softCam.jrPusherAxisZ.downPos.inPos )
      Coil( "Unit1.Em7.ControlNodes".jellyRollWinder."step".transition1[1120] )
   END_RUNG
   RUNG wire#w1
      Contact( "Unit1.Em7.ControlNodes".jellyRollWinder."step".transition1[1120] )
      Move(in := #JOB_11_STEP_90, out1 => "Unit1.Em7.ControlNodes".jellyRollWinder.sequence.status.nextStep)
   END_RUNG
   // the same network as SCL:
   #_w1 := ("Unit1.Em7.ControlNodes".jellyRollWinder.sequence.status.currentStep = #JOB_11_STEP_20) AND "Unit1.Em7.ControlNodes".jellyRollWinder.sequence.status.seqActive;
   "Unit1.Em7.ControlNodes".jellyRollWinder."step".action1[1120] := #_w1 AND NOT "Unit1.Em7.ControlNodes".cm.softCam.jrPusherAxisZ.downPos.inPos;
   "Unit1.Em7.ControlNodes".jellyRollWinder."step".transition1[1120] := #_w1 AND "Unit1.Em7.ControlNodes".cm.softCam.jrPusherAxisZ.downPos.inPos;
   IF #_w1 AND "Unit1.Em7.ControlNodes".jellyRollWinder."step".transition1[1120] THEN
       "Unit1.Em7.ControlNodes".jellyRollWinder.sequence.status.nextStep := #JOB_11_STEP_90;
   END_IF;
END_REGION

REGION Network 54: Step[1190] : Job[11] Step End
   RUNG wire#powerrail
      { S7_Templates := "SrcType := DInt" } EQ_Contact(in1 := "Unit1.Em7.ControlNodes".jellyRollWinder.sequence.status.currentStep, in2 := #JOB_11_STEP_90)
      Contact( "Unit1.Em7.ControlNodes".jellyRollWinder.sequence.status.seqActive )
      wire#w1
      Coil( "Unit1.Em7.ControlNodes".jellyRollWinder."step".action1[1190] )
   END_RUNG
   RUNG wire#w1
      Coil( "Unit1.Em7.ControlNodes".jellyRollWinder."step".transition1[1190] )
   END_RUNG
   RUNG wire#w1
      Contact( "Unit1.Em7.ControlNodes".jellyRollWinder."step".transition1[1190] )
      Move(in := #STEP_IDLE, out1 => "Unit1.Em7.ControlNodes".jellyRollWinder.sequence.status.nextStep)
   END_RUNG
   // the same network as SCL:
   "Unit1.Em7.ControlNodes".jellyRollWinder."step".action1[1190] := ("Unit1.Em7.ControlNodes".jellyRollWinder.sequence.status.currentStep = #JOB_11_STEP_90) AND "Unit1.Em7.ControlNodes".jellyRollWinder.sequence.status.seqActive;
   "Unit1.Em7.ControlNodes".jellyRollWinder."step".transition1[1190] := ("Unit1.Em7.ControlNodes".jellyRollWinder.sequence.status.currentStep = #JOB_11_STEP_90) AND "Unit1.Em7.ControlNodes".jellyRollWinder.sequence.status.seqActive;
   IF ("Unit1.Em7.ControlNodes".jellyRollWinder.sequence.status.currentStep = #JOB_11_STEP_90) AND "Unit1.Em7.ControlNodes".jellyRollWinder.sequence.status.seqActive AND "Unit1.Em7.ControlNodes".jellyRollWinder."step".transition1[1190] THEN
       "Unit1.Em7.ControlNodes".jellyRollWinder.sequence.status.nextStep := #STEP_IDLE;
   END_IF;
END_REGION

REGION Network 55: *************** JOB[12] Cam StartSync ************************
END_REGION

REGION Network 56: Step[1201] : JOB[12] Condition
   RUNG wire#powerrail
      { S7_Templates := "SrcType := DInt" } EQ_Contact(in1 := "Unit1.Em7.ControlNodes".jellyRollWinder.sequence.status.currentStep, in2 := #JOB_12_STEP_01)
      Contact( "Unit1.Em7.ControlNodes".jellyRollWinder.sequence.status.seqActive )
      wire#w1
      Coil( "Unit1.Em7.ControlNodes".jellyRollWinder."step".action1[1201] )
   END_RUNG
   RUNG wire#w1
      Coil( "Unit1.Em7.ControlNodes".jellyRollWinder."step".transition1[1201] )
   END_RUNG
   RUNG wire#w1
      Contact( "Unit1.Em7.ControlNodes".jellyRollWinder."step".transition1[1201] )
      Move(in := #JOB_12_STEP_10, out1 => "Unit1.Em7.ControlNodes".jellyRollWinder.sequence.status.nextStep)
   END_RUNG
   // the same network as SCL:
   "Unit1.Em7.ControlNodes".jellyRollWinder."step".action1[1201] := ("Unit1.Em7.ControlNodes".jellyRollWinder.sequence.status.currentStep = #JOB_12_STEP_01) AND "Unit1.Em7.ControlNodes".jellyRollWinder.sequence.status.seqActive;
   "Unit1.Em7.ControlNodes".jellyRollWinder."step".transition1[1201] := ("Unit1.Em7.ControlNodes".jellyRollWinder.sequence.status.currentStep = #JOB_12_STEP_01) AND "Unit1.Em7.ControlNodes".jellyRollWinder.sequence.status.seqActive;
   IF ("Unit1.Em7.ControlNodes".jellyRollWinder.sequence.status.currentStep = #JOB_12_STEP_01) AND "Unit1.Em7.ControlNodes".jellyRollWinder.sequence.status.seqActive AND "Unit1.Em7.ControlNodes".jellyRollWinder."step".transition1[1201] THEN
       "Unit1.Em7.ControlNodes".jellyRollWinder.sequence.status.nextStep := #JOB_12_STEP_10;
   END_IF;
END_REGION

REGION Network 57: Step[1210] : Pusher Z-Axis Cam Calculate
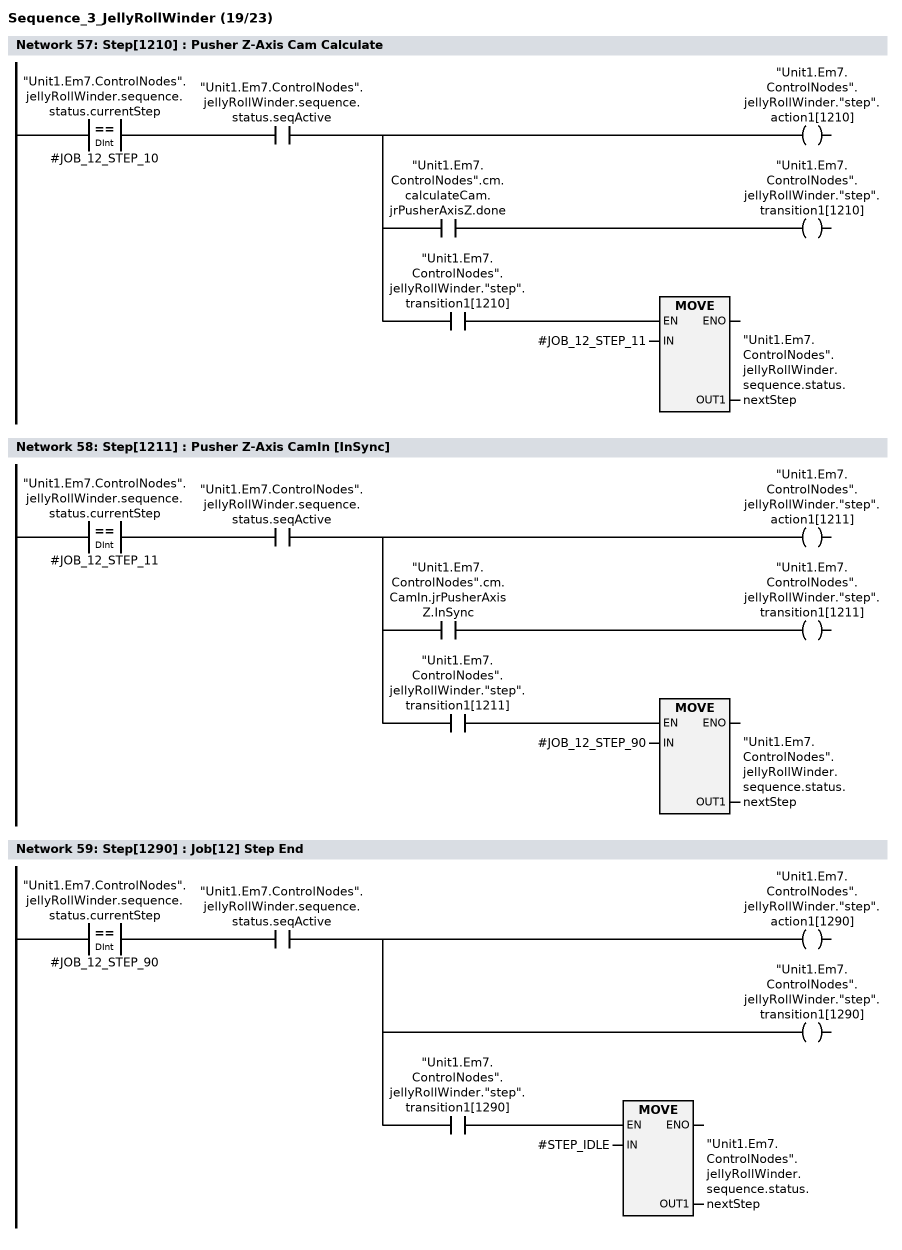
   RUNG wire#powerrail
      { S7_Templates := "SrcType := DInt" } EQ_Contact(in1 := "Unit1.Em7.ControlNodes".jellyRollWinder.sequence.status.currentStep, in2 := #JOB_12_STEP_10)
      Contact( "Unit1.Em7.ControlNodes".jellyRollWinder.sequence.status.seqActive )
      wire#w1
      Coil( "Unit1.Em7.ControlNodes".jellyRollWinder."step".action1[1210] )
   END_RUNG
   RUNG wire#w1
      Contact( "Unit1.Em7.ControlNodes".cm.calculateCam.jrPusherAxisZ.done )
      Coil( "Unit1.Em7.ControlNodes".jellyRollWinder."step".transition1[1210] )
   END_RUNG
   RUNG wire#w1
      Contact( "Unit1.Em7.ControlNodes".jellyRollWinder."step".transition1[1210] )
      Move(in := #JOB_12_STEP_11, out1 => "Unit1.Em7.ControlNodes".jellyRollWinder.sequence.status.nextStep)
   END_RUNG
   // the same network as SCL:
   "Unit1.Em7.ControlNodes".jellyRollWinder."step".action1[1210] := ("Unit1.Em7.ControlNodes".jellyRollWinder.sequence.status.currentStep = #JOB_12_STEP_10) AND "Unit1.Em7.ControlNodes".jellyRollWinder.sequence.status.seqActive;
   "Unit1.Em7.ControlNodes".jellyRollWinder."step".transition1[1210] := ("Unit1.Em7.ControlNodes".jellyRollWinder.sequence.status.currentStep = #JOB_12_STEP_10) AND "Unit1.Em7.ControlNodes".jellyRollWinder.sequence.status.seqActive AND "Unit1.Em7.ControlNodes".cm.calculateCam.jrPusherAxisZ.done;
   IF ("Unit1.Em7.ControlNodes".jellyRollWinder.sequence.status.currentStep = #JOB_12_STEP_10) AND "Unit1.Em7.ControlNodes".jellyRollWinder.sequence.status.seqActive AND "Unit1.Em7.ControlNodes".jellyRollWinder."step".transition1[1210] THEN
       "Unit1.Em7.ControlNodes".jellyRollWinder.sequence.status.nextStep := #JOB_12_STEP_11;
   END_IF;
END_REGION

REGION Network 58: Step[1211] : Pusher Z-Axis CamIn [InSync]
   RUNG wire#powerrail
      { S7_Templates := "SrcType := DInt" } EQ_Contact(in1 := "Unit1.Em7.ControlNodes".jellyRollWinder.sequence.status.currentStep, in2 := #JOB_12_STEP_11)
      Contact( "Unit1.Em7.ControlNodes".jellyRollWinder.sequence.status.seqActive )
      wire#w1
      Coil( "Unit1.Em7.ControlNodes".jellyRollWinder."step".action1[1211] )
   END_RUNG
   RUNG wire#w1
      Contact( "Unit1.Em7.ControlNodes".cm.CamIn.jrPusherAxisZ.InSync )
      Coil( "Unit1.Em7.ControlNodes".jellyRollWinder."step".transition1[1211] )
   END_RUNG
   RUNG wire#w1
      Contact( "Unit1.Em7.ControlNodes".jellyRollWinder."step".transition1[1211] )
      Move(in := #JOB_12_STEP_90, out1 => "Unit1.Em7.ControlNodes".jellyRollWinder.sequence.status.nextStep)
   END_RUNG
   // the same network as SCL:
   "Unit1.Em7.ControlNodes".jellyRollWinder."step".action1[1211] := ("Unit1.Em7.ControlNodes".jellyRollWinder.sequence.status.currentStep = #JOB_12_STEP_11) AND "Unit1.Em7.ControlNodes".jellyRollWinder.sequence.status.seqActive;
   "Unit1.Em7.ControlNodes".jellyRollWinder."step".transition1[1211] := ("Unit1.Em7.ControlNodes".jellyRollWinder.sequence.status.currentStep = #JOB_12_STEP_11) AND "Unit1.Em7.ControlNodes".jellyRollWinder.sequence.status.seqActive AND "Unit1.Em7.ControlNodes".cm.CamIn.jrPusherAxisZ.InSync;
   IF ("Unit1.Em7.ControlNodes".jellyRollWinder.sequence.status.currentStep = #JOB_12_STEP_11) AND "Unit1.Em7.ControlNodes".jellyRollWinder.sequence.status.seqActive AND "Unit1.Em7.ControlNodes".jellyRollWinder."step".transition1[1211] THEN
       "Unit1.Em7.ControlNodes".jellyRollWinder.sequence.status.nextStep := #JOB_12_STEP_90;
   END_IF;
END_REGION

REGION Network 59: Step[1290] : Job[12] Step End
   RUNG wire#powerrail
      { S7_Templates := "SrcType := DInt" } EQ_Contact(in1 := "Unit1.Em7.ControlNodes".jellyRollWinder.sequence.status.currentStep, in2 := #JOB_12_STEP_90)
      Contact( "Unit1.Em7.ControlNodes".jellyRollWinder.sequence.status.seqActive )
      wire#w1
      Coil( "Unit1.Em7.ControlNodes".jellyRollWinder."step".action1[1290] )
   END_RUNG
   RUNG wire#w1
      Coil( "Unit1.Em7.ControlNodes".jellyRollWinder."step".transition1[1290] )
   END_RUNG
   RUNG wire#w1
      Contact( "Unit1.Em7.ControlNodes".jellyRollWinder."step".transition1[1290] )
      Move(in := #STEP_IDLE, out1 => "Unit1.Em7.ControlNodes".jellyRollWinder.sequence.status.nextStep)
   END_RUNG
   // the same network as SCL:
   "Unit1.Em7.ControlNodes".jellyRollWinder."step".action1[1290] := ("Unit1.Em7.ControlNodes".jellyRollWinder.sequence.status.currentStep = #JOB_12_STEP_90) AND "Unit1.Em7.ControlNodes".jellyRollWinder.sequence.status.seqActive;
   "Unit1.Em7.ControlNodes".jellyRollWinder."step".transition1[1290] := ("Unit1.Em7.ControlNodes".jellyRollWinder.sequence.status.currentStep = #JOB_12_STEP_90) AND "Unit1.Em7.ControlNodes".jellyRollWinder.sequence.status.seqActive;
   IF ("Unit1.Em7.ControlNodes".jellyRollWinder.sequence.status.currentStep = #JOB_12_STEP_90) AND "Unit1.Em7.ControlNodes".jellyRollWinder.sequence.status.seqActive AND "Unit1.Em7.ControlNodes".jellyRollWinder."step".transition1[1290] THEN
       "Unit1.Em7.ControlNodes".jellyRollWinder.sequence.status.nextStep := #STEP_IDLE;
   END_IF;
END_REGION

REGION Network 60: *************** JOB[13] Cam 2nd Widning ************************
END_REGION

